LIN {X 0,Y 474.686,Z 291.355,A -85,B 0,C 180,E1 -7407.334,E2 -7407.334} C_VEL
LIN {X 0,Y 474.609,Z 291.36,A -85,B 0,C 180,E1 -7410.23,E2 -7410.23} C_VEL
LIN {X 0,Y 474.639,Z 291.365,A -85,B 0,C 180,E1 -7413.22,E2 -7413.22} C_VEL
LIN {X 0,Y 474.588,Z 291.363,A -85,B 0,C 180,E1 -7416.323,E2 -7416.323} C_VEL
LIN {X 0,Y 474.631,Z 291.363,A -85,B 0,C 180,E1 -7419.647,E2 -7419.647} C_VEL
LIN {X 0,Y 474.618,Z 291.361,A -85,B 0,C 180,E1 -7422.934,E2 -7422.934} C_VEL
LIN {X 0,Y 474.609,Z 291.365,A -85,B 0,C 180,E1 -7425.894,E2 -7425.894} C_VEL
LIN {X 0,Y 474.631,Z 291.358,A -85,B 0,C 180,E1 -7429.04,E2 -7429.04} C_VEL
LIN {X 0,Y 474.613,Z 291.367,A -85,B 0,C 180,E1 -7431.703,E2 -7431.703} C_VEL
LIN {X 0,Y 474.628,Z 291.358,A -85,B 0,C 180,E1 -7434.725,E2 -7434.725} C_VEL
LIN {X 0,Y 474.639,Z 291.362,A -85,B 0,C 180,E1 -7437.787,E2 -7437.787} C_VEL
LIN {X 0,Y 474.627,Z 291.358,A -85,B 0,C 180,E1 -7440.884,E2 -7440.884} C_VEL
LIN {X 0,Y 474.657,Z 291.356,A -85,B 0,C 180,E1 -7443.627,E2 -7443.627} C_VEL
LIN {X 0,Y 474.638,Z 291.36,A -85,B 0,C 180,E1 -7446.641,E2 -7446.641} C_VEL
LIN {X 0,Y 474.658,Z 291.358,A -85,B 0,C 180,E1 -7450.089,E2 -7450.089} C_VEL
LIN {X 0,Y 474.657,Z 291.354,A -85,B 0,C 180,E1 -7451.665,E2 -7451.665} C_VEL
LIN {X 0,Y 473.993,Z 291.444,A -85,B 0,C 180,E1 -7452.374,E2 -7452.374} C_VEL
LIN {X 0,Y 471.142,Z 291.796,A -85,B 0,C 180,E1 -7453.526,E2 -7453.526} C_VEL
LIN {X 0,Y 468.727,Z 292.1,A -85,B 0,C 180,E1 -7454.454,E2 -7454.454} C_VEL
LIN {X 0,Y 467.686,Z 292.224,A -85,B 0,C 180,E1 -7455.171,E2 -7455.171} C_VEL
LIN {X 0,Y 467.599,Z 292.234,A -85,B 0,C 180,E1 -7455.414,E2 -7455.414} C_VEL
LIN {X 0,Y 467.653,Z 292.235,A -85,B 0,C 180,E1 -7458.733,E2 -7458.733} C_VEL
LIN {X 0,Y 467.671,Z 292.229,A -85,B 0,C 180,E1 -7461.356,E2 -7461.356} C_VEL
LIN {X 0,Y 467.766,Z 292.344,A -85,B 0,C 180,E1 -7464.313,E2 -7464.313} C_VEL
LIN {X 0,Y 468.704,Z 298.944,A -85,B 0,C 180,E1 -7465.699,E2 -7465.699} C_VEL
LIN {X 0,Y 468.406,Z 311.043,A -85,B 0,C 180,E1 -7468.104,E2 -7468.104} C_VEL
LIN {X 0,Y 471.308,Z 326.851,A -85,B 0,C 180,E1 -7468.452,E2 -7468.452} C_VEL
LIN {X 0,Y 470.486,Z 418.039,A -85,B 0,C 180,E1 -7469.865,E2 -7469.865} C_VEL
LIN {X 0,Y 470.214,Z 431.176,A -85,B 0,C 180,E1 -7470.24,E2 -7470.24} C_VEL
LIN {X 0,Y 469.922,Z 444.292,A -85,B 0,C 180,E1 -7470.802,E2 -7470.802} C_VEL
LIN {X 0,Y 469.502,Z 456.173,A -85,B 0,C 180,E1 -7471.5,E2 -7471.5} C_VEL
LIN {X 0,Y 468.934,Z 467.583,A -85,B 0,C 180,E1 -7472.361,E2 -7472.361} C_VEL
LIN {X 0,Y 468.432,Z 477.859,A -85,B 0,C 180,E1 -7473.332,E2 -7473.332} C_VEL
LIN {X 0,Y 468.034,Z 486.265,A -85,B 0,C 180,E1 -7474.304,E2 -7474.304} C_VEL
LIN {X 0,Y 467.605,Z 495.387,A -85,B 0,C 180,E1 -7475.605,E2 -7475.605} C_VEL
LIN {X 0,Y 467.327,Z 503.183,A -85,B 0,C 180,E1 -7476.996,E2 -7476.996} C_VEL
LIN {X 0,Y 467.054,Z 508.653,A -85,B 0,C 180,E1 -7478.217,E2 -7478.217} C_VEL
LIN {X 0,Y 466.859,Z 513.329,A -85,B 0,C 180,E1 -7479.53,E2 -7479.53} C_VEL
LIN {X 0,Y 466.774,Z 516.89,A -85,B 0,C 180,E1 -7480.847,E2 -7480.847} C_VEL
LIN {X 0,Y 466.656,Z 519.437,A -85,B 0,C 180,E1 -7482.17,E2 -7482.17} C_VEL
LIN {X 0,Y 466.575,Z 520.608,A -85,B 0,C 180,E1 -7483.057,E2 -7483.057} C_VEL
LIN {X 0,Y 466.55,Z 521.33,A -85,B 0,C 180,E1 -7483.945,E2 -7483.945} C_VEL
LIN {X 0,Y 466.612,Z 521.631,A -85,B 0,C 180,E1 -7485.431,E2 -7485.431} C_VEL
LIN {X 0,Y 466.524,Z 521.04,A -85,B 0,C 180,E1 -7486.631,E2 -7486.631} C_VEL
LIN {X 0,Y 466.586,Z 520.075,A -85,B 0,C 180,E1 -7487.531,E2 -7487.531} C_VEL
LIN {X 0,Y 466.672,Z 518.689,A -85,B 0,C 180,E1 -7488.435,E2 -7488.435} C_VEL
LIN {X 0,Y 466.786,Z 515.7,A -85,B 0,C 180,E1 -7489.8,E2 -7489.8} C_VEL
LIN {X 0,Y 466.941,Z 511.554,A -85,B 0,C 180,E1 -7491.174,E2 -7491.174} C_VEL
LIN {X 0,Y 467.176,Z 506.077,A -85,B 0,C 180,E1 -7492.556,E2 -7492.556} C_VEL
LIN {X 0,Y 467.518,Z 499.072,A -85,B 0,C 180,E1 -7493.945,E2 -7493.945} C_VEL
LIN {X 0,Y 467.901,Z 491.826,A -85,B 0,C 180,E1 -7495.106,E2 -7495.106} C_VEL
LIN {X 0,Y 468.344,Z 482.951,A -85,B 0,C 180,E1 -7496.273,E2 -7496.273} C_VEL
LIN {X 0,Y 468.855,Z 473.048,A -85,B 0,C 180,E1 -7497.325,E2 -7497.325} C_VEL
LIN {X 0,Y 469.363,Z 461.573,A -85,B 0,C 180,E1 -7498.3,E2 -7498.3} C_VEL
LIN {X 0,Y 469.901,Z 449.823,A -85,B 0,C 180,E1 -7499.081,E2 -7499.081} C_VEL
LIN {X 0,Y 470.273,Z 438.126,A -85,B 0,C 180,E1 -7499.671,E2 -7499.671} C_VEL
LIN {X 0,Y 470.613,Z 424.916,A -85,B 0,C 180,E1 -7500.145,E2 -7500.145} C_VEL
LIN {X 0,Y 470.839,Z 411.912,A -85,B 0,C 180,E1 -7500.431,E2 -7500.431} C_VEL
LIN {X 0,Y 471.52,Z 325.739,A -85,B 0,C 180,E1 -7501.764,E2 -7501.764} C_VEL
LIN {X 0,Y 468.523,Z 310.731,A -85,B 0,C 180,E1 -7502.149,E2 -7502.149} C_VEL
LIN {X 0,Y 468.717,Z 298.947,A -85,B 0,C 180,E1 -7504.445,E2 -7504.445} C_VEL
LIN {X 0,Y 467.528,Z 292.25,A -85,B 0,C 180,E1 -7505.833,E2 -7505.833} C_VEL
LIN {X 0,Y 467.53,Z 292.248,A -85,B 0,C 180,E1 -7509.148,E2 -7509.148} C_VEL
LIN {X 0,Y 467.547,Z 292.247,A -85,B 0,C 180,E1 -7511.404,E2 -7511.404} C_VEL
LIN {X 0,Y 467.552,Z 292.246,A -85,B 0,C 180,E1 -7515.051,E2 -7515.051} C_VEL
LIN {X 0,Y 467.55,Z 292.242,A -85,B 0,C 180,E1 -7518.724,E2 -7518.724} C_VEL
LIN {X 0,Y 467.53,Z 292.248,A -85,B 0,C 180,E1 -7521.952,E2 -7521.952} C_VEL
LIN {X 0,Y 467.54,Z 292.236,A -85,B 0,C 180,E1 -7525.165,E2 -7525.165} C_VEL
LIN {X 0,Y 467.569,Z 292.238,A -85,B 0,C 180,E1 -7528.259,E2 -7528.259} C_VEL
LIN {X 0,Y 467.54,Z 292.244,A -85,B 0,C 180,E1 -7531.248,E2 -7531.248} C_VEL
LIN {X 0,Y 467.565,Z 292.241,A -85,B 0,C 180,E1 -7534.158,E2 -7534.158} C_VEL
LIN {X 0,Y 467.561,Z 292.239,A -85,B 0,C 180,E1 -7536.995,E2 -7536.995} C_VEL
LIN {X 0,Y 467.607,Z 292.234,A -85,B 0,C 180,E1 -7539.777,E2 -7539.777} C_VEL
LIN {X 0,Y 467.581,Z 292.236,A -85,B 0,C 180,E1 -7542.506,E2 -7542.506} C_VEL
LIN {X 0,Y 467.586,Z 292.236,A -85,B 0,C 180,E1 -7545.196,E2 -7545.196} C_VEL
LIN {X 0,Y 467.641,Z 292.231,A -85,B 0,C 180,E1 -7547.854,E2 -7547.854} C_VEL
LIN {X 0,Y 467.666,Z 292.226,A -85,B 0,C 180,E1 -7551.357,E2 -7551.357} C_VEL
LIN {X 0,Y 467.705,Z 292.219,A -85,B 0,C 180,E1 -7553.962,E2 -7553.962} C_VEL
LIN {X 0,Y 467.843,Z 292.2,A -85,B 0,C 180,E1 -7557.417,E2 -7557.417} C_VEL
LIN {X 0,Y 467.865,Z 292.201,A -85,B 0,C 180,E1 -7560,E2 -7560} C_VEL
LIN {X 0,Y 467.844,Z 292.205,A -85,B 0,C 180,E1 -7562.583,E2 -7562.583} C_VEL
LIN {X 0,Y 467.721,Z 292.22,A -85,B 0,C 180,E1 -7566.038,E2 -7566.038} C_VEL
LIN {X 0,Y 467.668,Z 292.226,A -85,B 0,C 180,E1 -7568.643,E2 -7568.643} C_VEL
LIN {X 0,Y 467.643,Z 292.229,A -85,B 0,C 180,E1 -7572.146,E2 -7572.146} C_VEL
LIN {X 0,Y 467.625,Z 292.231,A -85,B 0,C 180,E1 -7575.696,E2 -7575.696} C_VEL
LIN {X 0,Y 467.604,Z 292.235,A -85,B 0,C 180,E1 -7578.765,E2 -7578.765} C_VEL
LIN {X 0,Y 467.568,Z 292.243,A -85,B 0,C 180,E1 -7581.269,E2 -7581.269} C_VEL
LIN {X 0,Y 467.56,Z 292.236,A -85,B 0,C 180,E1 -7583.944,E2 -7583.944} C_VEL
LIN {X 0,Y 467.616,Z 292.237,A -85,B 0,C 180,E1 -7586.801,E2 -7586.801} C_VEL
LIN {X 0,Y 467.577,Z 292.24,A -85,B 0,C 180,E1 -7589.737,E2 -7589.737} C_VEL
LIN {X 0,Y 467.573,Z 292.237,A -85,B 0,C 180,E1 -7592.759,E2 -7592.759} C_VEL
LIN {X 0,Y 467.547,Z 292.243,A -85,B 0,C 180,E1 -7595.891,E2 -7595.891} C_VEL
LIN {X 0,Y 467.607,Z 292.239,A -85,B 0,C 180,E1 -7599.143,E2 -7599.143} C_VEL
LIN {X 0,Y 467.577,Z 292.237,A -85,B 0,C 180,E1 -7602.568,E2 -7602.568} C_VEL
LIN {X 0,Y 467.563,Z 292.24,A -85,B 0,C 180,E1 -7605.055,E2 -7605.055} C_VEL
LIN {X 0,Y 467.617,Z 292.235,A -85,B 0,C 180,E1 -7607.445,E2 -7607.445} C_VEL
LIN {X 0,Y 467.593,Z 292.234,A -85,B 0,C 180,E1 -7610.859,E2 -7610.859} C_VEL
LIN {X 0,Y 467.557,Z 292.245,A -85,B 0,C 180,E1 -7614.262,E2 -7614.262} C_VEL
LIN {X 0,Y 467.577,Z 292.24,A -85,B 0,C 180,E1 -7617.322,E2 -7617.322} C_VEL
LIN {X 0,Y 467.566,Z 292.242,A -85,B 0,C 180,E1 -7620.669,E2 -7620.669} C_VEL
LIN {X 0,Y 467.651,Z 292.234,A -85,B 0,C 180,E1 -7623.805,E2 -7623.805} C_VEL
LIN {X 0,Y 469.721,Z 302.869,A -85,B 0,C 180,E1 -7625.88,E2 -7625.88} C_VEL
LIN {X 0,Y 469.887,Z 307.145,A -85,B 0,C 180,E1 -7626.651,E2 -7626.651} C_VEL
LIN {X 0,Y 469.041,Z 325.461,A -85,B 0,C 180,E1 -7629.843,E2 -7629.843} C_VEL
LIN {X 0,Y 468.324,Z 343.295,A -85,B 0,C 180,E1 -7632.901,E2 -7632.901} C_VEL
LIN {X 0,Y 471.288,Z 362.293,A -85,B 0,C 180,E1 -7633.33,E2 -7633.33} C_VEL
LIN {X 0,Y 470.632,Z 452.171,A -85,B 0,C 180,E1 -7634.742,E2 -7634.742} C_VEL
LIN {X 0,Y 470.231,Z 465.287,A -85,B 0,C 180,E1 -7635.116,E2 -7635.116} C_VEL
LIN {X 0,Y 469.711,Z 477.936,A -85,B 0,C 180,E1 -7635.653,E2 -7635.653} C_VEL
LIN {X 0,Y 469.259,Z 489.997,A -85,B 0,C 180,E1 -7636.358,E2 -7636.358} C_VEL
LIN {X 0,Y 468.677,Z 501.749,A -85,B 0,C 180,E1 -7637.243,E2 -7637.243} C_VEL
LIN {X 0,Y 468.177,Z 512.937,A -85,B 0,C 180,E1 -7638.309,E2 -7638.309} C_VEL
LIN {X 0,Y 467.726,Z 522.081,A -85,B 0,C 180,E1 -7639.395,E2 -7639.395} C_VEL
LIN {X 0,Y 467.289,Z 531.006,A -85,B 0,C 180,E1 -7640.697,E2 -7640.697} C_VEL
LIN {X 0,Y 467.01,Z 538.19,A -85,B 0,C 180,E1 -7642,E2 -7642} C_VEL
LIN {X 0,Y 466.858,Z 543.046,A -85,B 0,C 180,E1 -7643.084,E2 -7643.084} C_VEL
LIN {X 0,Y 466.76,Z 547.769,A -85,B 0,C 180,E1 -7644.385,E2 -7644.385} C_VEL
LIN {X 0,Y 466.647,Z 551.376,A -85,B 0,C 180,E1 -7645.683,E2 -7645.683} C_VEL
LIN {X 0,Y 466.689,Z 553.239,A -85,B 0,C 180,E1 -7646.548,E2 -7646.548} C_VEL
LIN {X 0,Y 466.661,Z 554.634,A -85,B 0,C 180,E1 -7647.412,E2 -7647.412} C_VEL
LIN {X 0,Y 466.619,Z 556.239,A -85,B 0,C 180,E1 -7649.138,E2 -7649.138} C_VEL
LIN {X 0,Y 466.601,Z 556.45,A -85,B 0,C 180,E1 -7650.001,E2 -7650.001} C_VEL
LIN {X 0,Y 466.619,Z 556.229,A -85,B 0,C 180,E1 -7650.864,E2 -7650.864} C_VEL
LIN {X 0,Y 466.662,Z 554.617,A -85,B 0,C 180,E1 -7652.591,E2 -7652.591} C_VEL
LIN {X 0,Y 466.69,Z 553.208,A -85,B 0,C 180,E1 -7653.455,E2 -7653.455} C_VEL
LIN {X 0,Y 466.69,Z 550.25,A -85,B 0,C 180,E1 -7654.752,E2 -7654.752} C_VEL
LIN {X 0,Y 466.752,Z 546.245,A -85,B 0,C 180,E1 -7656.051,E2 -7656.051} C_VEL
LIN {X 0,Y 466.944,Z 540.078,A -85,B 0,C 180,E1 -7657.569,E2 -7657.569} C_VEL
LIN {X 0,Y 467.176,Z 533.344,A -85,B 0,C 180,E1 -7658.871,E2 -7658.871} C_VEL
LIN {X 0,Y 467.504,Z 524.988,A -85,B 0,C 180,E1 -7660.175,E2 -7660.175} C_VEL
LIN {X 0,Y 467.954,Z 516.396,A -85,B 0,C 180,E1 -7661.26,E2 -7661.26} C_VEL
LIN {X 0,Y 468.443,Z 506.232,A -85,B 0,C 180,E1 -7662.304,E2 -7662.304} C_VEL
LIN {X 0,Y 468.889,Z 495.273,A -85,B 0,C 180,E1 -7663.214,E2 -7663.214} C_VEL
LIN {X 0,Y 469.398,Z 483.688,A -85,B 0,C 180,E1 -7663.972,E2 -7663.972} C_VEL
LIN {X 0,Y 469.845,Z 471.654,A -85,B 0,C 180,E1 -7664.566,E2 -7664.566} C_VEL
LIN {X 0,Y 470.282,Z 458.632,A -85,B 0,C 180,E1 -7665.023,E2 -7665.023} C_VEL
LIN {X 0,Y 470.471,Z 446.371,A -85,B 0,C 180,E1 -7665.294,E2 -7665.294} C_VEL
LIN {X 0,Y 471.081,Z 362.542,A -85,B 0,C 180,E1 -7666.579,E2 -7666.579} C_VEL
LIN {X 0,Y 468.245,Z 343.636,A -85,B 0,C 180,E1 -7666.969,E2 -7666.969} C_VEL
LIN {X 0,Y 468.944,Z 326.257,A -85,B 0,C 180,E1 -7669.936,E2 -7669.936} C_VEL
LIN {X 0,Y 469.786,Z 306.459,A -85,B 0,C 180,E1 -7673.357,E2 -7673.357} C_VEL
LIN {X 0,Y 469.594,Z 302.376,A -85,B 0,C 180,E1 -7674.085,E2 -7674.085} C_VEL
LIN {X 0,Y 467.65,Z 292.236,A -85,B 0,C 180,E1 -7676.018,E2 -7676.018} C_VEL
LIN {X 0,Y 467.58,Z 292.239,A -85,B 0,C 180,E1 -7678.75,E2 -7678.75} C_VEL
LIN {X 0,Y 467.588,Z 292.237,A -85,B 0,C 180,E1 -7681.741,E2 -7681.741} C_VEL
LIN {X 0,Y 467.564,Z 292.24,A -85,B 0,C 180,E1 -7684.834,E2 -7684.834} C_VEL
LIN {X 0,Y 467.57,Z 292.241,A -85,B 0,C 180,E1 -7688.045,E2 -7688.045} C_VEL
LIN {X 0,Y 467.584,Z 292.236,A -85,B 0,C 180,E1 -7691.277,E2 -7691.277} C_VEL
LIN {X 0,Y 467.555,Z 292.239,A -85,B 0,C 180,E1 -7693.821,E2 -7693.821} C_VEL
LIN {X 0,Y 467.56,Z 292.241,A -85,B 0,C 180,E1 -7696.256,E2 -7696.256} C_VEL
LIN {X 0,Y 467.584,Z 292.244,A -85,B 0,C 180,E1 -7698.724,E2 -7698.724} C_VEL
LIN {X 0,Y 467.57,Z 292.237,A -85,B 0,C 180,E1 -7701.956,E2 -7701.956} C_VEL
LIN {X 0,Y 467.564,Z 292.244,A -85,B 0,C 180,E1 -7705.167,E2 -7705.167} C_VEL
LIN {X 0,Y 467.584,Z 292.235,A -85,B 0,C 180,E1 -7708.26,E2 -7708.26} C_VEL
LIN {X 0,Y 467.583,Z 292.243,A -85,B 0,C 180,E1 -7711.251,E2 -7711.251} C_VEL
LIN {X 0,Y 467.607,Z 292.232,A -85,B 0,C 180,E1 -7714.16,E2 -7714.16} C_VEL
LIN {X 0,Y 467.583,Z 292.239,A -85,B 0,C 180,E1 -7716.996,E2 -7716.996} C_VEL
LIN {X 0,Y 467.628,Z 292.234,A -85,B 0,C 180,E1 -7719.777,E2 -7719.777} C_VEL
LIN {X 0,Y 467.603,Z 292.233,A -85,B 0,C 180,E1 -7722.506,E2 -7722.506} C_VEL
LIN {X 0,Y 467.611,Z 292.235,A -85,B 0,C 180,E1 -7725.196,E2 -7725.196} C_VEL
LIN {X 0,Y 467.662,Z 292.232,A -85,B 0,C 180,E1 -7727.855,E2 -7727.855} C_VEL
LIN {X 0,Y 467.684,Z 292.225,A -85,B 0,C 180,E1 -7731.357,E2 -7731.357} C_VEL
LIN {X 0,Y 467.725,Z 292.226,A -85,B 0,C 180,E1 -7733.962,E2 -7733.962} C_VEL
LIN {X 0,Y 467.863,Z 292.202,A -85,B 0,C 180,E1 -7737.417,E2 -7737.417} C_VEL
LIN {X 0,Y 467.885,Z 292.205,A -85,B 0,C 180,E1 -7740,E2 -7740} C_VEL
LIN {X 0,Y 467.862,Z 292.204,A -85,B 0,C 180,E1 -7742.583,E2 -7742.583} C_VEL
LIN {X 0,Y 467.738,Z 292.221,A -85,B 0,C 180,E1 -7746.037,E2 -7746.037} C_VEL
LIN {X 0,Y 467.674,Z 292.229,A -85,B 0,C 180,E1 -7748.643,E2 -7748.643} C_VEL
LIN {X 0,Y 467.661,Z 292.229,A -85,B 0,C 180,E1 -7752.145,E2 -7752.145} C_VEL
LIN {X 0,Y 467.644,Z 292.228,A -85,B 0,C 180,E1 -7755.695,E2 -7755.695} C_VEL
LIN {X 0,Y 467.627,Z 292.232,A -85,B 0,C 180,E1 -7759.307,E2 -7759.307} C_VEL
LIN {X 0,Y 467.539,Z 292.241,A -85,B 0,C 180,E1 -7762.073,E2 -7762.073} C_VEL
LIN {X 0,Y 467.608,Z 292.241,A -85,B 0,C 180,E1 -7764.887,E2 -7764.887} C_VEL
LIN {X 0,Y 467.625,Z 292.231,A -85,B 0,C 180,E1 -7767.769,E2 -7767.769} C_VEL
LIN {X 0,Y 467.572,Z 292.245,A -85,B 0,C 180,E1 -7771.044,E2 -7771.044} C_VEL
LIN {X 0,Y 467.592,Z 292.234,A -85,B 0,C 180,E1 -7774.242,E2 -7774.242} C_VEL
LIN {X 0,Y 467.547,Z 292.247,A -85,B 0,C 180,E1 -7777.185,E2 -7777.185} C_VEL
LIN {X 0,Y 467.582,Z 292.236,A -85,B 0,C 180,E1 -7780.264,E2 -7780.264} C_VEL
LIN {X 0,Y 467.591,Z 292.234,A -85,B 0,C 180,E1 -7782.566,E2 -7782.566} C_VEL
LIN {X 0,Y 467.57,Z 292.239,A -85,B 0,C 180,E1 -7785.052,E2 -7785.052} C_VEL
LIN {X 0,Y 467.593,Z 292.24,A -85,B 0,C 180,E1 -7787.439,E2 -7787.439} C_VEL
LIN {X 0,Y 467.563,Z 292.238,A -85,B 0,C 180,E1 -7790.852,E2 -7790.852} C_VEL
LIN {X 0,Y 467.563,Z 292.241,A -85,B 0,C 180,E1 -7794.26,E2 -7794.26} C_VEL
LIN {X 0,Y 467.585,Z 292.236,A -85,B 0,C 180,E1 -7797.32,E2 -7797.32} C_VEL
LIN {X 0,Y 467.573,Z 292.238,A -85,B 0,C 180,E1 -7800.667,E2 -7800.667} C_VEL
LIN {X 0,Y 467.616,Z 292.231,A -85,B 0,C 180,E1 -7803.199,E2 -7803.199} C_VEL
LIN {X 0,Y 467.594,Z 292.24,A -85,B 0,C 180,E1 -7806.468,E2 -7806.468} C_VEL
LIN {X 0,Y 467.626,Z 292.231,A -85,B 0,C 180,E1 -7809.776,E2 -7809.776} C_VEL
LIN {X 0,Y 467.609,Z 292.241,A -85,B 0,C 180,E1 -7812.506,E2 -7812.506} C_VEL
LIN {X 0,Y 467.599,Z 292.234,A -85,B 0,C 180,E1 -7815.414,E2 -7815.414} C_VEL
LIN {X 0,Y 466.928,Z 292.321,A -85,B 0,C 180,E1 -7816.133,E2 -7816.133} C_VEL
LIN {X 0,Y 464.085,Z 292.673,A -85,B 0,C 180,E1 -7817.302,E2 -7817.302} C_VEL
LIN {X 0,Y 461.686,Z 292.973,A -85,B 0,C 180,E1 -7818.244,E2 -7818.244} C_VEL
LIN {X 0,Y 460.658,Z 293.103,A -85,B 0,C 180,E1 -7818.971,E2 -7818.971} C_VEL
LIN {X 0,Y 460.576,Z 293.109,A -85,B 0,C 180,E1 -7819.218,E2 -7819.218} C_VEL
LIN {X 0,Y 460.691,Z 293.102,A -85,B 0,C 180,E1 -7822.566,E2 -7822.566} C_VEL
LIN {X 0,Y 460.698,Z 293.153,A -85,B 0,C 180,E1 -7824.143,E2 -7824.143} C_VEL
LIN {X 0,Y 461.745,Z 300.164,A -85,B 0,C 180,E1 -7825.634,E2 -7825.634} C_VEL
LIN {X 0,Y 461.437,Z 311.165,A -85,B 0,C 180,E1 -7827.862,E2 -7827.862} C_VEL
LIN {X 0,Y 464.399,Z 326.503,A -85,B 0,C 180,E1 -7828.211,E2 -7828.211} C_VEL
LIN {X 0,Y 463.6,Z 418.943,A -85,B 0,C 180,E1 -7829.673,E2 -7829.673} C_VEL
LIN {X 0,Y 463.311,Z 431.88,A -85,B 0,C 180,E1 -7830.053,E2 -7830.053} C_VEL
LIN {X 0,Y 463.032,Z 444.33,A -85,B 0,C 180,E1 -7830.597,E2 -7830.597} C_VEL
LIN {X 0,Y 462.583,Z 456.292,A -85,B 0,C 180,E1 -7831.305,E2 -7831.305} C_VEL
LIN {X 0,Y 462.007,Z 467.734,A -85,B 0,C 180,E1 -7832.178,E2 -7832.178} C_VEL
LIN {X 0,Y 461.453,Z 478.048,A -85,B 0,C 180,E1 -7833.164,E2 -7833.164} C_VEL
LIN {X 0,Y 461.033,Z 486.476,A -85,B 0,C 180,E1 -7834.151,E2 -7834.151} C_VEL
LIN {X 0,Y 460.586,Z 495.616,A -85,B 0,C 180,E1 -7835.471,E2 -7835.471} C_VEL
LIN {X 0,Y 460.29,Z 502.846,A -85,B 0,C 180,E1 -7836.769,E2 -7836.769} C_VEL
LIN {X 0,Y 460.059,Z 507.991,A -85,B 0,C 180,E1 -7837.901,E2 -7837.901} C_VEL
LIN {X 0,Y 459.81,Z 512.864,A -85,B 0,C 180,E1 -7839.234,E2 -7839.234} C_VEL
LIN {X 0,Y 459.718,Z 516.605,A -85,B 0,C 180,E1 -7840.569,E2 -7840.569} C_VEL
LIN {X 0,Y 459.621,Z 519.256,A -85,B 0,C 180,E1 -7841.871,E2 -7841.871} C_VEL
LIN {X 0,Y 459.481,Z 521.074,A -85,B 0,C 180,E1 -7843.262,E2 -7843.262} C_VEL
LIN {X 0,Y 459.469,Z 521.716,A -85,B 0,C 180,E1 -7844.165,E2 -7844.165} C_VEL
LIN {X 0,Y 459.52,Z 521.884,A -85,B 0,C 180,E1 -7845.521,E2 -7845.521} C_VEL
LIN {X 0,Y 459.449,Z 521.102,A -85,B 0,C 180,E1 -7846.894,E2 -7846.894} C_VEL
LIN {X 0,Y 459.599,Z 518.882,A -85,B 0,C 180,E1 -7848.545,E2 -7848.545} C_VEL
LIN {X 0,Y 459.761,Z 515.355,A -85,B 0,C 180,E1 -7850.115,E2 -7850.115} C_VEL
LIN {X 0,Y 459.921,Z 510.995,A -85,B 0,C 180,E1 -7851.513,E2 -7851.513} C_VEL
LIN {X 0,Y 460.209,Z 505.305,A -85,B 0,C 180,E1 -7852.917,E2 -7852.917} C_VEL
LIN {X 0,Y 460.573,Z 498.069,A -85,B 0,C 180,E1 -7854.329,E2 -7854.329} C_VEL
LIN {X 0,Y 461.048,Z 489.45,A -85,B 0,C 180,E1 -7855.659,E2 -7855.659} C_VEL
LIN {X 0,Y 461.547,Z 480.205,A -85,B 0,C 180,E1 -7856.813,E2 -7856.813} C_VEL
LIN {X 0,Y 462.05,Z 470.897,A -85,B 0,C 180,E1 -7857.761,E2 -7857.761} C_VEL
LIN {X 0,Y 462.608,Z 459.799,A -85,B 0,C 180,E1 -7858.676,E2 -7858.676} C_VEL
LIN {X 0,Y 463.136,Z 448.139,A -85,B 0,C 180,E1 -7859.423,E2 -7859.423} C_VEL
LIN {X 0,Y 463.549,Z 435.864,A -85,B 0,C 180,E1 -7860.019,E2 -7860.019} C_VEL
LIN {X 0,Y 463.847,Z 423.53,A -85,B 0,C 180,E1 -7860.442,E2 -7860.442} C_VEL
LIN {X 0,Y 464.086,Z 408.879,A -85,B 0,C 180,E1 -7860.734,E2 -7860.734} C_VEL
LIN {X 0,Y 464.733,Z 326.376,A -85,B 0,C 180,E1 -7862.032,E2 -7862.032} C_VEL
LIN {X 0,Y 461.613,Z 310.999,A -85,B 0,C 180,E1 -7862.439,E2 -7862.439} C_VEL
LIN {X 0,Y 461.704,Z 299.479,A -85,B 0,C 180,E1 -7864.717,E2 -7864.717} C_VEL
LIN {X 0,Y 460.466,Z 293.13,A -85,B 0,C 180,E1 -7866.084,E2 -7866.084} C_VEL
LIN {X 0,Y 460.479,Z 293.126,A -85,B 0,C 180,E1 -7868.888,E2 -7868.888} C_VEL
LIN {X 0,Y 460.49,Z 293.127,A -85,B 0,C 180,E1 -7871.597,E2 -7871.597} C_VEL
LIN {X 0,Y 460.499,Z 293.121,A -85,B 0,C 180,E1 -7874.588,E2 -7874.588} C_VEL
LIN {X 0,Y 460.478,Z 293.127,A -85,B 0,C 180,E1 -7877.814,E2 -7877.814} C_VEL
LIN {X 0,Y 460.497,Z 293.122,A -85,B 0,C 180,E1 -7880.134,E2 -7880.134} C_VEL
LIN {X 0,Y 460.451,Z 293.126,A -85,B 0,C 180,E1 -7883.468,E2 -7883.468} C_VEL
LIN {X 0,Y 460.506,Z 293.119,A -85,B 0,C 180,E1 -7886.673,E2 -7886.673} C_VEL
LIN {X 0,Y 460.494,Z 293.126,A -85,B 0,C 180,E1 -7889.759,E2 -7889.759} C_VEL
LIN {X 0,Y 460.518,Z 293.117,A -85,B 0,C 180,E1 -7892.753,E2 -7892.753} C_VEL
LIN {X 0,Y 460.508,Z 293.12,A -85,B 0,C 180,E1 -7895.666,E2 -7895.666} C_VEL
LIN {X 0,Y 460.507,Z 293.115,A -85,B 0,C 180,E1 -7898.578,E2 -7898.578} C_VEL
LIN {X 0,Y 460.571,Z 293.111,A -85,B 0,C 180,E1 -7901.31,E2 -7901.31} C_VEL
LIN {X 0,Y 460.589,Z 293.11,A -85,B 0,C 180,E1 -7904.059,E2 -7904.059} C_VEL
LIN {X 0,Y 460.594,Z 293.107,A -85,B 0,C 180,E1 -7907.666,E2 -7907.666} C_VEL
LIN {X 0,Y 460.613,Z 293.104,A -85,B 0,C 180,E1 -7911.224,E2 -7911.224} C_VEL
LIN {X 0,Y 460.669,Z 293.094,A -85,B 0,C 180,E1 -7913.87,E2 -7913.87} C_VEL
LIN {X 0,Y 460.785,Z 293.079,A -85,B 0,C 180,E1 -7917.378,E2 -7917.378} C_VEL
LIN {X 0,Y 460.836,Z 293.077,A -85,B 0,C 180,E1 -7920,E2 -7920} C_VEL
LIN {X 0,Y 460.785,Z 293.083,A -85,B 0,C 180,E1 -7922.623,E2 -7922.623} C_VEL
LIN {X 0,Y 460.687,Z 293.097,A -85,B 0,C 180,E1 -7926.13,E2 -7926.13} C_VEL
LIN {X 0,Y 460.615,Z 293.105,A -85,B 0,C 180,E1 -7928.777,E2 -7928.777} C_VEL
LIN {X 0,Y 460.599,Z 293.109,A -85,B 0,C 180,E1 -7932.445,E2 -7932.445} C_VEL
LIN {X 0,Y 460.586,Z 293.108,A -85,B 0,C 180,E1 -7935.998,E2 -7935.998} C_VEL
LIN {X 0,Y 460.557,Z 293.113,A -85,B 0,C 180,E1 -7938.902,E2 -7938.902} C_VEL
LIN {X 0,Y 460.503,Z 293.12,A -85,B 0,C 180,E1 -7941.486,E2 -7941.486} C_VEL
LIN {X 0,Y 460.53,Z 293.112,A -85,B 0,C 180,E1 -7944.333,E2 -7944.333} C_VEL
LIN {X 0,Y 460.572,Z 293.112,A -85,B 0,C 180,E1 -7947.244,E2 -7947.244} C_VEL
LIN {X 0,Y 460.519,Z 293.117,A -85,B 0,C 180,E1 -7950.24,E2 -7950.24} C_VEL
LIN {X 0,Y 460.519,Z 293.123,A -85,B 0,C 180,E1 -7953.326,E2 -7953.326} C_VEL
LIN {X 0,Y 460.47,Z 293.122,A -85,B 0,C 180,E1 -7956.53,E2 -7956.53} C_VEL
LIN {X 0,Y 460.567,Z 293.115,A -85,B 0,C 180,E1 -7959.859,E2 -7959.859} C_VEL
LIN {X 0,Y 460.508,Z 293.118,A -85,B 0,C 180,E1 -7962.902,E2 -7962.902} C_VEL
LIN {X 0,Y 460.516,Z 293.115,A -85,B 0,C 180,E1 -7965.83,E2 -7965.83} C_VEL
LIN {X 0,Y 460.536,Z 293.116,A -85,B 0,C 180,E1 -7968.992,E2 -7968.992} C_VEL
LIN {X 0,Y 460.533,Z 293.116,A -85,B 0,C 180,E1 -7971.27,E2 -7971.27} C_VEL
LIN {X 0,Y 460.507,Z 293.121,A -85,B 0,C 180,E1 -7974.556,E2 -7974.556} C_VEL
LIN {X 0,Y 460.526,Z 293.123,A -85,B 0,C 180,E1 -7977.717,E2 -7977.717} C_VEL
LIN {X 0,Y 460.536,Z 293.118,A -85,B 0,C 180,E1 -7980.771,E2 -7980.771} C_VEL
LIN {X 0,Y 460.622,Z 293.272,A -85,B 0,C 180,E1 -7983.618,E2 -7983.618} C_VEL
LIN {X 0,Y 462.827,Z 304.413,A -85,B 0,C 180,E1 -7985.797,E2 -7985.797} C_VEL
LIN {X 0,Y 462.972,Z 308.34,A -85,B 0,C 180,E1 -7986.519,E2 -7986.519} C_VEL
LIN {X 0,Y 462.08,Z 326.655,A -85,B 0,C 180,E1 -7989.758,E2 -7989.758} C_VEL
LIN {X 0,Y 461.369,Z 343.062,A -85,B 0,C 180,E1 -7992.62,E2 -7992.62} C_VEL
LIN {X 0,Y 464.544,Z 363.97,A -85,B 0,C 180,E1 -7993.089,E2 -7993.089} C_VEL
LIN {X 0,Y 463.843,Z 451.619,A -85,B 0,C 180,E1 -7994.485,E2 -7994.485} C_VEL
LIN {X 0,Y 463.429,Z 464.827,A -85,B 0,C 180,E1 -7994.865,E2 -7994.865} C_VEL
LIN {X 0,Y 462.86,Z 478.082,A -85,B 0,C 180,E1 -7995.436,E2 -7995.436} C_VEL
LIN {X 0,Y 462.367,Z 490.017,A -85,B 0,C 180,E1 -7996.15,E2 -7996.15} C_VEL
LIN {X 0,Y 461.792,Z 500.723,A -85,B 0,C 180,E1 -7996.965,E2 -7996.965} C_VEL
LIN {X 0,Y 461.28,Z 511.808,A -85,B 0,C 180,E1 -7998.02,E2 -7998.02} C_VEL
LIN {X 0,Y 460.794,Z 520.272,A -85,B 0,C 180,E1 -7999.011,E2 -7999.011} C_VEL
LIN {X 0,Y 460.309,Z 529.459,A -85,B 0,C 180,E1 -8000.333,E2 -8000.333} C_VEL
LIN {X 0,Y 460,Z 536.87,A -85,B 0,C 180,E1 -8001.656,E2 -8001.656} C_VEL
LIN {X 0,Y 459.775,Z 542.83,A -85,B 0,C 180,E1 -8002.977,E2 -8002.977} C_VEL
LIN {X 0,Y 459.656,Z 547.542,A -85,B 0,C 180,E1 -8004.298,E2 -8004.298} C_VEL
LIN {X 0,Y 459.564,Z 551.141,A -85,B 0,C 180,E1 -8005.616,E2 -8005.616} C_VEL
LIN {X 0,Y 459.585,Z 552.995,A -85,B 0,C 180,E1 -8006.494,E2 -8006.494} C_VEL
LIN {X 0,Y 459.584,Z 554.385,A -85,B 0,C 180,E1 -8007.372,E2 -8007.372} C_VEL
LIN {X 0,Y 459.523,Z 555.981,A -85,B 0,C 180,E1 -8009.125,E2 -8009.125} C_VEL
LIN {X 0,Y 459.532,Z 556.186,A -85,B 0,C 180,E1 -8010.001,E2 -8010.001} C_VEL
LIN {X 0,Y 459.552,Z 555.958,A -85,B 0,C 180,E1 -8010.878,E2 -8010.878} C_VEL
LIN {X 0,Y 459.584,Z 554.336,A -85,B 0,C 180,E1 -8012.631,E2 -8012.631} C_VEL
LIN {X 0,Y 459.586,Z 552.917,A -85,B 0,C 180,E1 -8013.508,E2 -8013.508} C_VEL
LIN {X 0,Y 459.617,Z 549.951,A -85,B 0,C 180,E1 -8014.826,E2 -8014.826} C_VEL
LIN {X 0,Y 459.716,Z 544.886,A -85,B 0,C 180,E1 -8016.432,E2 -8016.432} C_VEL
LIN {X 0,Y 459.894,Z 538.732,A -85,B 0,C 180,E1 -8017.907,E2 -8017.907} C_VEL
LIN {X 0,Y 460.189,Z 531.755,A -85,B 0,C 180,E1 -8019.229,E2 -8019.229} C_VEL
LIN {X 0,Y 460.564,Z 523.002,A -85,B 0,C 180,E1 -8020.552,E2 -8020.552} C_VEL
LIN {X 0,Y 461.058,Z 514.04,A -85,B 0,C 180,E1 -8021.654,E2 -8021.654} C_VEL
LIN {X 0,Y 461.546,Z 504.309,A -85,B 0,C 180,E1 -8022.633,E2 -8022.633} C_VEL
LIN {X 0,Y 462.016,Z 493.31,A -85,B 0,C 180,E1 -8023.527,E2 -8023.527} C_VEL
LIN {X 0,Y 462.576,Z 481.107,A -85,B 0,C 180,E1 -8024.295,E2 -8024.295} C_VEL
LIN {X 0,Y 463.048,Z 468.338,A -85,B 0,C 180,E1 -8024.898,E2 -8024.898} C_VEL
LIN {X 0,Y 463.478,Z 455.671,A -85,B 0,C 180,E1 -8025.305,E2 -8025.305} C_VEL
LIN {X 0,Y 463.709,Z 439.528,A -85,B 0,C 180,E1 -8025.607,E2 -8025.607} C_VEL
LIN {X 0,Y 464.125,Z 362.39,A -85,B 0,C 180,E1 -8026.811,E2 -8026.811} C_VEL
LIN {X 0,Y 461.259,Z 343.25,A -85,B 0,C 180,E1 -8027.234,E2 -8027.234} C_VEL
LIN {X 0,Y 461.936,Z 327.178,A -85,B 0,C 180,E1 -8030.019,E2 -8030.019} C_VEL
LIN {X 0,Y 462.828,Z 307.357,A -85,B 0,C 180,E1 -8033.492,E2 -8033.492} C_VEL
LIN {X 0,Y 462.539,Z 303.123,A -85,B 0,C 180,E1 -8034.263,E2 -8034.263} C_VEL
LIN {X 0,Y 460.594,Z 293.114,A -85,B 0,C 180,E1 -8036.202,E2 -8036.202} C_VEL
LIN {X 0,Y 460.544,Z 293.115,A -85,B 0,C 180,E1 -8039.232,E2 -8039.232} C_VEL
LIN {X 0,Y 460.536,Z 293.121,A -85,B 0,C 180,E1 -8042.285,E2 -8042.285} C_VEL
LIN {X 0,Y 460.514,Z 293.116,A -85,B 0,C 180,E1 -8045.446,E2 -8045.446} C_VEL
LIN {X 0,Y 460.538,Z 293.115,A -85,B 0,C 180,E1 -8048.896,E2 -8048.896} C_VEL
LIN {X 0,Y 460.529,Z 293.118,A -85,B 0,C 180,E1 -8052.182,E2 -8052.182} C_VEL
LIN {X 0,Y 460.52,Z 293.116,A -85,B 0,C 180,E1 -8055.411,E2 -8055.411} C_VEL
LIN {X 0,Y 460.538,Z 293.117,A -85,B 0,C 180,E1 -8058.398,E2 -8058.398} C_VEL
LIN {X 0,Y 460.529,Z 293.117,A -85,B 0,C 180,E1 -8061.267,E2 -8061.267} C_VEL
LIN {X 0,Y 460.514,Z 293.119,A -85,B 0,C 180,E1 -8064.554,E2 -8064.554} C_VEL
LIN {X 0,Y 460.531,Z 293.115,A -85,B 0,C 180,E1 -8067.715,E2 -8067.715} C_VEL
LIN {X 0,Y 460.546,Z 293.116,A -85,B 0,C 180,E1 -8070.769,E2 -8070.769} C_VEL
LIN {X 0,Y 460.565,Z 293.112,A -85,B 0,C 180,E1 -8073.735,E2 -8073.735} C_VEL
LIN {X 0,Y 460.552,Z 293.112,A -85,B 0,C 180,E1 -8076.624,E2 -8076.624} C_VEL
LIN {X 0,Y 460.557,Z 293.119,A -85,B 0,C 180,E1 -8079.453,E2 -8079.453} C_VEL
LIN {X 0,Y 460.554,Z 293.112,A -85,B 0,C 180,E1 -8082.23,E2 -8082.23} C_VEL
LIN {X 0,Y 460.57,Z 293.11,A -85,B 0,C 180,E1 -8084.965,E2 -8084.965} C_VEL
LIN {X 0,Y 460.615,Z 293.104,A -85,B 0,C 180,E1 -8088.559,E2 -8088.559} C_VEL
LIN {X 0,Y 460.672,Z 293.101,A -85,B 0,C 180,E1 -8092.108,E2 -8092.108} C_VEL
LIN {X 0,Y 460.693,Z 293.094,A -85,B 0,C 180,E1 -8094.748,E2 -8094.748} C_VEL
LIN {X 0,Y 460.804,Z 293.081,A -85,B 0,C 180,E1 -8097.377,E2 -8097.377} C_VEL
LIN {X 0,Y 460.856,Z 293.081,A -85,B 0,C 180,E1 -8100,E2 -8100} C_VEL
LIN {X 0,Y 460.803,Z 293.083,A -85,B 0,C 180,E1 -8102.622,E2 -8102.622} C_VEL
LIN {X 0,Y 460.703,Z 293.099,A -85,B 0,C 180,E1 -8106.13,E2 -8106.13} C_VEL
LIN {X 0,Y 460.624,Z 293.106,A -85,B 0,C 180,E1 -8108.776,E2 -8108.776} C_VEL
LIN {X 0,Y 460.619,Z 293.111,A -85,B 0,C 180,E1 -8112.445,E2 -8112.445} C_VEL
LIN {X 0,Y 460.606,Z 293.106,A -85,B 0,C 180,E1 -8115.997,E2 -8115.997} C_VEL
LIN {X 0,Y 460.573,Z 293.109,A -85,B 0,C 180,E1 -8119.615,E2 -8119.615} C_VEL
LIN {X 0,Y 460.515,Z 293.119,A -85,B 0,C 180,E1 -8122.428,E2 -8122.428} C_VEL
LIN {X 0,Y 460.573,Z 293.109,A -85,B 0,C 180,E1 -8125.801,E2 -8125.801} C_VEL
LIN {X 0,Y 460.557,Z 293.111,A -85,B 0,C 180,E1 -8128.232,E2 -8128.232} C_VEL
LIN {X 0,Y 460.525,Z 293.121,A -85,B 0,C 180,E1 -8131.282,E2 -8131.282} C_VEL
LIN {X 0,Y 460.535,Z 293.114,A -85,B 0,C 180,E1 -8134.505,E2 -8134.505} C_VEL
LIN {X 0,Y 460.503,Z 293.122,A -85,B 0,C 180,E1 -8137.623,E2 -8137.623} C_VEL
LIN {X 0,Y 460.546,Z 293.112,A -85,B 0,C 180,E1 -8140.269,E2 -8140.269} C_VEL
LIN {X 0,Y 460.503,Z 293.124,A -85,B 0,C 180,E1 -8143.375,E2 -8143.375} C_VEL
LIN {X 0,Y 460.5,Z 293.118,A -85,B 0,C 180,E1 -8146.624,E2 -8146.624} C_VEL
LIN {X 0,Y 460.543,Z 293.122,A -85,B 0,C 180,E1 -8149.73,E2 -8149.73} C_VEL
LIN {X 0,Y 460.503,Z 293.118,A -85,B 0,C 180,E1 -8152.523,E2 -8152.523} C_VEL
LIN {X 0,Y 460.55,Z 293.116,A -85,B 0,C 180,E1 -8155.623,E2 -8155.623} C_VEL
LIN {X 0,Y 460.541,Z 293.113,A -85,B 0,C 180,E1 -8158.744,E2 -8158.744} C_VEL
LIN {X 0,Y 460.585,Z 293.115,A -85,B 0,C 180,E1 -8162.253,E2 -8162.253} C_VEL
LIN {X 0,Y 460.543,Z 293.115,A -85,B 0,C 180,E1 -8164.703,E2 -8164.703} C_VEL
LIN {X 0,Y 460.514,Z 293.116,A -85,B 0,C 180,E1 -8167.57,E2 -8167.57} C_VEL
LIN {X 0,Y 460.572,Z 293.117,A -85,B 0,C 180,E1 -8170.384,E2 -8170.384} C_VEL
LIN {X 0,Y 460.566,Z 293.111,A -85,B 0,C 180,E1 -8173.145,E2 -8173.145} C_VEL
LIN {X 0,Y 460.556,Z 293.111,A -85,B 0,C 180,E1 -8175.867,E2 -8175.867} C_VEL
LIN {X 0,Y 460.612,Z 293.111,A -85,B 0,C 180,E1 -8178.558,E2 -8178.558} C_VEL
LIN {X 0,Y 460.576,Z 293.109,A -85,B 0,C 180,E1 -8179.218,E2 -8179.218} C_VEL
LIN {X 0,Y 459.916,Z 293.191,A -85,B 0,C 180,E1 -8179.948,E2 -8179.948} C_VEL
LIN {X 0,Y 457.089,Z 293.549,A -85,B 0,C 180,E1 -8181.133,E2 -8181.133} C_VEL
LIN {X 0,Y 454.706,Z 293.85,A -85,B 0,C 180,E1 -8182.09,E2 -8182.09} C_VEL
LIN {X 0,Y 453.695,Z 293.975,A -85,B 0,C 180,E1 -8182.829,E2 -8182.829} C_VEL
LIN {X 0,Y 453.619,Z 293.983,A -85,B 0,C 180,E1 -8183.079,E2 -8183.079} C_VEL
LIN {X 0,Y 453.663,Z 294.077,A -85,B 0,C 180,E1 -8183.996,E2 -8183.996} C_VEL
LIN {X 0,Y 454.767,Z 301.367,A -85,B 0,C 180,E1 -8185.567,E2 -8185.567} C_VEL
LIN {X 0,Y 454.5,Z 311.383,A -85,B 0,C 180,E1 -8187.614,E2 -8187.614} C_VEL
LIN {X 0,Y 457.625,Z 327.961,A -85,B 0,C 180,E1 -8187.996,E2 -8187.996} C_VEL
LIN {X 0,Y 456.735,Z 418.419,A -85,B 0,C 180,E1 -8189.439,E2 -8189.439} C_VEL
LIN {X 0,Y 456.425,Z 431.394,A -85,B 0,C 180,E1 -8189.817,E2 -8189.817} C_VEL
LIN {X 0,Y 456.126,Z 444.366,A -85,B 0,C 180,E1 -8190.385,E2 -8190.385} C_VEL
LIN {X 0,Y 455.675,Z 456.387,A -85,B 0,C 180,E1 -8191.103,E2 -8191.103} C_VEL
LIN {X 0,Y 455.064,Z 467.864,A -85,B 0,C 180,E1 -8191.99,E2 -8191.99} C_VEL
LIN {X 0,Y 454.49,Z 478.199,A -85,B 0,C 180,E1 -8192.99,E2 -8192.99} C_VEL
LIN {X 0,Y 454.053,Z 486.645,A -85,B 0,C 180,E1 -8193.993,E2 -8193.993} C_VEL
LIN {X 0,Y 453.648,Z 494.445,A -85,B 0,C 180,E1 -8195.109,E2 -8195.109} C_VEL
LIN {X 0,Y 453.289,Z 502.321,A -85,B 0,C 180,E1 -8196.504,E2 -8196.504} C_VEL
LIN {X 0,Y 452.946,Z 509.119,A -85,B 0,C 180,E1 -8198.026,E2 -8198.026} C_VEL
LIN {X 0,Y 452.721,Z 513.812,A -85,B 0,C 180,E1 -8199.38,E2 -8199.38} C_VEL
LIN {X 0,Y 452.635,Z 517.384,A -85,B 0,C 180,E1 -8200.737,E2 -8200.737} C_VEL
LIN {X 0,Y 452.531,Z 519.657,A -85,B 0,C 180,E1 -8201.926,E2 -8201.926} C_VEL
LIN {X 0,Y 452.386,Z 521.536,A -85,B 0,C 180,E1 -8203.474,E2 -8203.474} C_VEL
LIN {X 0,Y 452.376,Z 522.092,A -85,B 0,C 180,E1 -8204.391,E2 -8204.391} C_VEL
LIN {X 0,Y 452.418,Z 522.139,A -85,B 0,C 180,E1 -8205.608,E2 -8205.608} C_VEL
LIN {X 0,Y 452.373,Z 521.17,A -85,B 0,C 180,E1 -8207.167,E2 -8207.167} C_VEL
LIN {X 0,Y 452.526,Z 519.058,A -85,B 0,C 180,E1 -8208.672,E2 -8208.672} C_VEL
LIN {X 0,Y 452.657,Z 516.264,A -85,B 0,C 180,E1 -8209.971,E2 -8209.971} C_VEL
LIN {X 0,Y 452.816,Z 512.192,A -85,B 0,C 180,E1 -8211.371,E2 -8211.371} C_VEL
LIN {X 0,Y 453.104,Z 506.677,A -85,B 0,C 180,E1 -8212.814,E2 -8212.814} C_VEL
LIN {X 0,Y 453.514,Z 499.7,A -85,B 0,C 180,E1 -8214.244,E2 -8214.244} C_VEL
LIN {X 0,Y 453.926,Z 492.474,A -85,B 0,C 180,E1 -8215.443,E2 -8215.443} C_VEL
LIN {X 0,Y 454.482,Z 483.647,A -85,B 0,C 180,E1 -8216.642,E2 -8216.642} C_VEL
LIN {X 0,Y 455.019,Z 473.904,A -85,B 0,C 180,E1 -8217.716,E2 -8217.716} C_VEL
LIN {X 0,Y 455.598,Z 462.85,A -85,B 0,C 180,E1 -8218.692,E2 -8218.692} C_VEL
LIN {X 0,Y 456.215,Z 450.728,A -85,B 0,C 180,E1 -8219.533,E2 -8219.533} C_VEL
LIN {X 0,Y 456.65,Z 439.236,A -85,B 0,C 180,E1 -8220.138,E2 -8220.138} C_VEL
LIN {X 0,Y 457.018,Z 426.417,A -85,B 0,C 180,E1 -8220.621,E2 -8220.621} C_VEL
LIN {X 0,Y 457.269,Z 413.73,A -85,B 0,C 180,E1 -8220.923,E2 -8220.923} C_VEL
LIN {X 0,Y 457.975,Z 327.037,A -85,B 0,C 180,E1 -8222.313,E2 -8222.313} C_VEL
LIN {X 0,Y 454.708,Z 311.384,A -85,B 0,C 180,E1 -8222.717,E2 -8222.717} C_VEL
LIN {X 0,Y 454.884,Z 301.951,A -85,B 0,C 180,E1 -8224.594,E2 -8224.594} C_VEL
LIN {X 0,Y 453.427,Z 294.007,A -85,B 0,C 180,E1 -8226.295,E2 -8226.295} C_VEL
LIN {X 0,Y 453.429,Z 294.006,A -85,B 0,C 180,E1 -8229.454,E2 -8229.454} C_VEL
LIN {X 0,Y 453.424,Z 294.005,A -85,B 0,C 180,E1 -8231.928,E2 -8231.928} C_VEL
LIN {X 0,Y 453.469,Z 293.998,A -85,B 0,C 180,E1 -8235.471,E2 -8235.471} C_VEL
LIN {X 0,Y 453.439,Z 294.001,A -85,B 0,C 180,E1 -8238.205,E2 -8238.205} C_VEL
LIN {X 0,Y 453.426,Z 294.002,A -85,B 0,C 180,E1 -8240.801,E2 -8240.801} C_VEL
LIN {X 0,Y 453.433,Z 293.994,A -85,B 0,C 180,E1 -8243.915,E2 -8243.915} C_VEL
LIN {X 0,Y 453.465,Z 293.998,A -85,B 0,C 180,E1 -8247.15,E2 -8247.15} C_VEL
LIN {X 0,Y 453.453,Z 293.999,A -85,B 0,C 180,E1 -8250.267,E2 -8250.267} C_VEL
LIN {X 0,Y 453.454,Z 293.998,A -85,B 0,C 180,E1 -8253.291,E2 -8253.291} C_VEL
LIN {X 0,Y 453.48,Z 293.998,A -85,B 0,C 180,E1 -8256.238,E2 -8256.238} C_VEL
LIN {X 0,Y 453.467,Z 293.991,A -85,B 0,C 180,E1 -8259.117,E2 -8259.117} C_VEL
LIN {X 0,Y 453.488,Z 293.999,A -85,B 0,C 180,E1 -8261.944,E2 -8261.944} C_VEL
LIN {X 0,Y 453.522,Z 293.989,A -85,B 0,C 180,E1 -8264.726,E2 -8264.726} C_VEL
LIN {X 0,Y 453.544,Z 293.987,A -85,B 0,C 180,E1 -8268.379,E2 -8268.379} C_VEL
LIN {X 0,Y 453.577,Z 293.981,A -85,B 0,C 180,E1 -8271.087,E2 -8271.087} C_VEL
LIN {X 0,Y 453.635,Z 293.97,A -85,B 0,C 180,E1 -8273.774,E2 -8273.774} C_VEL
LIN {X 0,Y 453.729,Z 293.958,A -85,B 0,C 180,E1 -8277.337,E2 -8277.337} C_VEL
LIN {X 0,Y 453.807,Z 293.952,A -85,B 0,C 180,E1 -8280,E2 -8280} C_VEL
LIN {X 0,Y 453.73,Z 293.961,A -85,B 0,C 180,E1 -8282.664,E2 -8282.664} C_VEL
LIN {X 0,Y 453.655,Z 293.974,A -85,B 0,C 180,E1 -8286.226,E2 -8286.226} C_VEL
LIN {X 0,Y 453.579,Z 293.981,A -85,B 0,C 180,E1 -8288.914,E2 -8288.914} C_VEL
LIN {X 0,Y 453.549,Z 293.989,A -85,B 0,C 180,E1 -8292.529,E2 -8292.529} C_VEL
LIN {X 0,Y 453.531,Z 293.988,A -85,B 0,C 180,E1 -8296.197,E2 -8296.197} C_VEL
LIN {X 0,Y 453.507,Z 293.991,A -85,B 0,C 180,E1 -8299.041,E2 -8299.041} C_VEL
LIN {X 0,Y 453.464,Z 293.995,A -85,B 0,C 180,E1 -8301.837,E2 -8301.837} C_VEL
LIN {X 0,Y 453.502,Z 293.99,A -85,B 0,C 180,E1 -8304.735,E2 -8304.735} C_VEL
LIN {X 0,Y 453.527,Z 293.983,A -85,B 0,C 180,E1 -8307.962,E2 -8307.962} C_VEL
LIN {X 0,Y 453.473,Z 293.997,A -85,B 0,C 180,E1 -8310.76,E2 -8310.76} C_VEL
LIN {X 0,Y 453.467,Z 293.998,A -85,B 0,C 180,E1 -8313.914,E2 -8313.914} C_VEL
LIN {X 0,Y 453.462,Z 294.001,A -85,B 0,C 180,E1 -8317.189,E2 -8317.189} C_VEL
LIN {X 0,Y 453.522,Z 293.994,A -85,B 0,C 180,E1 -8319.447,E2 -8319.447} C_VEL
LIN {X 0,Y 453.459,Z 293.997,A -85,B 0,C 180,E1 -8322.996,E2 -8322.996} C_VEL
LIN {X 0,Y 453.469,Z 293.992,A -85,B 0,C 180,E1 -8325.782,E2 -8325.782} C_VEL
LIN {X 0,Y 453.489,Z 293.995,A -85,B 0,C 180,E1 -8328.213,E2 -8328.213} C_VEL
LIN {X 0,Y 453.52,Z 293.987,A -85,B 0,C 180,E1 -8330.79,E2 -8330.79} C_VEL
LIN {X 0,Y 453.451,Z 294,A -85,B 0,C 180,E1 -8333.919,E2 -8333.919} C_VEL
LIN {X 0,Y 453.478,Z 293.995,A -85,B 0,C 180,E1 -8337.153,E2 -8337.153} C_VEL
LIN {X 0,Y 453.471,Z 293.999,A -85,B 0,C 180,E1 -8340.27,E2 -8340.27} C_VEL
LIN {X 0,Y 453.587,Z 294.107,A -85,B 0,C 180,E1 -8343.347,E2 -8343.347} C_VEL
LIN {X 0,Y 455.857,Z 305.669,A -85,B 0,C 180,E1 -8345.65,E2 -8345.65} C_VEL
LIN {X 0,Y 456.085,Z 309.571,A -85,B 0,C 180,E1 -8346.383,E2 -8346.383} C_VEL
LIN {X 0,Y 455.159,Z 326.543,A -85,B 0,C 180,E1 -8349.436,E2 -8349.436} C_VEL
LIN {X 0,Y 454.434,Z 342.777,A -85,B 0,C 180,E1 -8352.315,E2 -8352.315} C_VEL
LIN {X 0,Y 457.745,Z 363.806,A -85,B 0,C 180,E1 -8352.806,E2 -8352.806} C_VEL
LIN {X 0,Y 457.037,Z 451.085,A -85,B 0,C 180,E1 -8354.219,E2 -8354.219} C_VEL
LIN {X 0,Y 456.597,Z 464.367,A -85,B 0,C 180,E1 -8354.604,E2 -8354.604} C_VEL
LIN {X 0,Y 456.08,Z 477.111,A -85,B 0,C 180,E1 -8355.158,E2 -8355.158} C_VEL
LIN {X 0,Y 455.544,Z 488.453,A -85,B 0,C 180,E1 -8355.825,E2 -8355.825} C_VEL
LIN {X 0,Y 454.861,Z 500.637,A -85,B 0,C 180,E1 -8356.757,E2 -8356.757} C_VEL
LIN {X 0,Y 454.325,Z 511.735,A -85,B 0,C 180,E1 -8357.834,E2 -8357.834} C_VEL
LIN {X 0,Y 453.699,Z 521.807,A -85,B 0,C 180,E1 -8359.063,E2 -8359.063} C_VEL
LIN {X 0,Y 453.199,Z 530.677,A -85,B 0,C 180,E1 -8360.405,E2 -8360.405} C_VEL
LIN {X 0,Y 452.903,Z 537.807,A -85,B 0,C 180,E1 -8361.749,E2 -8361.749} C_VEL
LIN {X 0,Y 452.634,Z 544.318,A -85,B 0,C 180,E1 -8363.315,E2 -8363.315} C_VEL
LIN {X 0,Y 452.563,Z 548.627,A -85,B 0,C 180,E1 -8364.655,E2 -8364.655} C_VEL
LIN {X 0,Y 452.486,Z 550.913,A -85,B 0,C 180,E1 -8365.547,E2 -8365.547} C_VEL
LIN {X 0,Y 452.481,Z 552.754,A -85,B 0,C 180,E1 -8366.439,E2 -8366.439} C_VEL
LIN {X 0,Y 452.507,Z 554.139,A -85,B 0,C 180,E1 -8367.331,E2 -8367.331} C_VEL
LIN {X 0,Y 452.43,Z 555.724,A -85,B 0,C 180,E1 -8369.111,E2 -8369.111} C_VEL
LIN {X 0,Y 452.465,Z 555.921,A -85,B 0,C 180,E1 -8370.001,E2 -8370.001} C_VEL
LIN {X 0,Y 452.457,Z 555.065,A -85,B 0,C 180,E1 -8371.782,E2 -8371.782} C_VEL
LIN {X 0,Y 452.508,Z 554.054,A -85,B 0,C 180,E1 -8372.672,E2 -8372.672} C_VEL
LIN {X 0,Y 452.484,Z 552.624,A -85,B 0,C 180,E1 -8373.563,E2 -8373.563} C_VEL
LIN {X 0,Y 452.546,Z 549.648,A -85,B 0,C 180,E1 -8374.901,E2 -8374.901} C_VEL
LIN {X 0,Y 452.612,Z 545.056,A -85,B 0,C 180,E1 -8376.397,E2 -8376.397} C_VEL
LIN {X 0,Y 452.842,Z 538.386,A -85,B 0,C 180,E1 -8378.03,E2 -8378.03} C_VEL
LIN {X 0,Y 453.13,Z 531.376,A -85,B 0,C 180,E1 -8379.374,E2 -8379.374} C_VEL
LIN {X 0,Y 453.543,Z 522.582,A -85,B 0,C 180,E1 -8380.718,E2 -8380.718} C_VEL
LIN {X 0,Y 454.133,Z 512.595,A -85,B 0,C 180,E1 -8381.947,E2 -8381.947} C_VEL
LIN {X 0,Y 454.642,Z 502.297,A -85,B 0,C 180,E1 -8382.965,E2 -8382.965} C_VEL
LIN {X 0,Y 455.152,Z 491.13,A -85,B 0,C 180,E1 -8383.848,E2 -8383.848} C_VEL
LIN {X 0,Y 455.732,Z 478.429,A -85,B 0,C 180,E1 -8384.628,E2 -8384.628} C_VEL
LIN {X 0,Y 456.189,Z 466.01,A -85,B 0,C 180,E1 -8385.184,E2 -8385.184} C_VEL
LIN {X 0,Y 456.652,Z 452.196,A -85,B 0,C 180,E1 -8385.597,E2 -8385.597} C_VEL
LIN {X 0,Y 457.409,Z 364.388,A -85,B 0,C 180,E1 -8387.007,E2 -8387.007} C_VEL
LIN {X 0,Y 454.263,Z 343.075,A -85,B 0,C 180,E1 -8387.467,E2 -8387.467} C_VEL
LIN {X 0,Y 454.983,Z 326.75,A -85,B 0,C 180,E1 -8390.339,E2 -8390.339} C_VEL
LIN {X 0,Y 455.883,Z 308.247,A -85,B 0,C 180,E1 -8393.631,E2 -8393.631} C_VEL
LIN {X 0,Y 455.467,Z 303.891,A -85,B 0,C 180,E1 -8394.44,E2 -8394.44} C_VEL
LIN {X 0,Y 453.551,Z 293.992,A -85,B 0,C 180,E1 -8396.377,E2 -8396.377} C_VEL
LIN {X 0,Y 453.514,Z 293.992,A -85,B 0,C 180,E1 -8398.713,E2 -8398.713} C_VEL
LIN {X 0,Y 453.469,Z 293.997,A -85,B 0,C 180,E1 -8401.8,E2 -8401.8} C_VEL
LIN {X 0,Y 453.482,Z 293.993,A -85,B 0,C 180,E1 -8404.99,E2 -8404.99} C_VEL
LIN {X 0,Y 453.465,Z 294.002,A -85,B 0,C 180,E1 -8408.313,E2 -8408.313} C_VEL
LIN {X 0,Y 453.5,Z 293.997,A -85,B 0,C 180,E1 -8410.609,E2 -8410.609} C_VEL
LIN {X 0,Y 453.459,Z 293.996,A -85,B 0,C 180,E1 -8413.244,E2 -8413.244} C_VEL
LIN {X 0,Y 453.469,Z 293.994,A -85,B 0,C 180,E1 -8415.779,E2 -8415.779} C_VEL
LIN {X 0,Y 453.485,Z 293.994,A -85,B 0,C 180,E1 -8418.21,E2 -8418.21} C_VEL
LIN {X 0,Y 453.497,Z 293.999,A -85,B 0,C 180,E1 -8420.794,E2 -8420.794} C_VEL
LIN {X 0,Y 453.46,Z 293.995,A -85,B 0,C 180,E1 -8423.917,E2 -8423.917} C_VEL
LIN {X 0,Y 453.48,Z 293.999,A -85,B 0,C 180,E1 -8427.151,E2 -8427.151} C_VEL
LIN {X 0,Y 453.481,Z 293.992,A -85,B 0,C 180,E1 -8430.268,E2 -8430.268} C_VEL
LIN {X 0,Y 453.511,Z 293.996,A -85,B 0,C 180,E1 -8433.294,E2 -8433.294} C_VEL
LIN {X 0,Y 453.508,Z 293.989,A -85,B 0,C 180,E1 -8436.239,E2 -8436.239} C_VEL
LIN {X 0,Y 453.488,Z 293.996,A -85,B 0,C 180,E1 -8439.118,E2 -8439.118} C_VEL
LIN {X 0,Y 453.509,Z 293.992,A -85,B 0,C 180,E1 -8441.944,E2 -8441.944} C_VEL
LIN {X 0,Y 453.545,Z 293.984,A -85,B 0,C 180,E1 -8444.726,E2 -8444.726} C_VEL
LIN {X 0,Y 453.564,Z 293.983,A -85,B 0,C 180,E1 -8448.379,E2 -8448.379} C_VEL
LIN {X 0,Y 453.595,Z 293.978,A -85,B 0,C 180,E1 -8451.086,E2 -8451.086} C_VEL
LIN {X 0,Y 453.655,Z 293.977,A -85,B 0,C 180,E1 -8453.774,E2 -8453.774} C_VEL
LIN {X 0,Y 453.748,Z 293.96,A -85,B 0,C 180,E1 -8457.337,E2 -8457.337} C_VEL
LIN {X 0,Y 453.826,Z 293.956,A -85,B 0,C 180,E1 -8460,E2 -8460} C_VEL
LIN {X 0,Y 453.747,Z 293.961,A -85,B 0,C 180,E1 -8462.663,E2 -8462.663} C_VEL
LIN {X 0,Y 453.67,Z 293.976,A -85,B 0,C 180,E1 -8466.225,E2 -8466.225} C_VEL
LIN {X 0,Y 453.59,Z 293.981,A -85,B 0,C 180,E1 -8468.913,E2 -8468.913} C_VEL
LIN {X 0,Y 453.569,Z 293.99,A -85,B 0,C 180,E1 -8472.529,E2 -8472.529} C_VEL
LIN {X 0,Y 453.55,Z 293.986,A -85,B 0,C 180,E1 -8476.196,E2 -8476.196} C_VEL
LIN {X 0,Y 453.522,Z 293.991,A -85,B 0,C 180,E1 -8479.039,E2 -8479.039} C_VEL
LIN {X 0,Y 453.481,Z 293.992,A -85,B 0,C 180,E1 -8481.836,E2 -8481.836} C_VEL
LIN {X 0,Y 453.518,Z 293.993,A -85,B 0,C 180,E1 -8484.734,E2 -8484.734} C_VEL
LIN {X 0,Y 453.537,Z 293.985,A -85,B 0,C 180,E1 -8487.959,E2 -8487.959} C_VEL
LIN {X 0,Y 453.47,Z 293.997,A -85,B 0,C 180,E1 -8491.524,E2 -8491.524} C_VEL
LIN {X 0,Y 453.491,Z 293.993,A -85,B 0,C 180,E1 -8494.777,E2 -8494.777} C_VEL
LIN {X 0,Y 453.467,Z 293.994,A -85,B 0,C 180,E1 -8498.311,E2 -8498.311} C_VEL
LIN {X 0,Y 453.498,Z 293.99,A -85,B 0,C 180,E1 -8500.608,E2 -8500.608} C_VEL
LIN {X 0,Y 453.459,Z 294,A -85,B 0,C 180,E1 -8503.243,E2 -8503.243} C_VEL
LIN {X 0,Y 453.466,Z 294,A -85,B 0,C 180,E1 -8505.778,E2 -8505.778} C_VEL
LIN {X 0,Y 453.483,Z 293.994,A -85,B 0,C 180,E1 -8508.209,E2 -8508.209} C_VEL
LIN {X 0,Y 453.491,Z 293.991,A -85,B 0,C 180,E1 -8510.794,E2 -8510.794} C_VEL
LIN {X 0,Y 453.458,Z 294.003,A -85,B 0,C 180,E1 -8513.916,E2 -8513.916} C_VEL
LIN {X 0,Y 453.486,Z 293.992,A -85,B 0,C 180,E1 -8517.15,E2 -8517.15} C_VEL
LIN {X 0,Y 453.479,Z 293.998,A -85,B 0,C 180,E1 -8520.267,E2 -8520.267} C_VEL
LIN {X 0,Y 453.505,Z 293.989,A -85,B 0,C 180,E1 -8523.293,E2 -8523.293} C_VEL
LIN {X 0,Y 453.501,Z 293.998,A -85,B 0,C 180,E1 -8526.238,E2 -8526.238} C_VEL
LIN {X 0,Y 453.485,Z 293.992,A -85,B 0,C 180,E1 -8529.117,E2 -8529.117} C_VEL
LIN {X 0,Y 453.513,Z 293.99,A -85,B 0,C 180,E1 -8531.943,E2 -8531.943} C_VEL
LIN {X 0,Y 453.542,Z 293.991,A -85,B 0,C 180,E1 -8534.725,E2 -8534.725} C_VEL
LIN {X 0,Y 453.561,Z 293.987,A -85,B 0,C 180,E1 -8538.378,E2 -8538.378} C_VEL
LIN {X 0,Y 453.587,Z 293.986,A -85,B 0,C 180,E1 -8541.085,E2 -8541.085} C_VEL
LIN {X 0,Y 453.619,Z 293.983,A -85,B 0,C 180,E1 -8543.079,E2 -8543.079} C_VEL
LIN {X 0,Y 453.352,Z 294.423,A -85,B 0,C 180,E1 -8543.569,E2 -8543.569} C_VEL
LIN {X 0,Y 452.663,Z 295.565,A -85,B 0,C 180,E1 -8544.037,E2 -8544.037} C_VEL
LIN {X 0,Y 450.63,Z 299.139,A -85,B 0,C 180,E1 -8544.908,E2 -8544.908} C_VEL
LIN {X 0,Y 448.557,Z 303.624,A -85,B 0,C 180,E1 -8545.749,E2 -8545.749} C_VEL
LIN {X 0,Y 447.668,Z 306.911,A -85,B 0,C 180,E1 -8546.392,E2 -8546.392} C_VEL
LIN {X 0,Y 447.598,Z 307.98,A -85,B 0,C 180,E1 -8546.611,E2 -8546.611} C_VEL
LIN {X 0,Y 447.538,Z 311.575,A -85,B 0,C 180,E1 -8547.354,E2 -8547.354} C_VEL
LIN {X 0,Y 450.828,Z 329.522,A -85,B 0,C 180,E1 -8547.782,E2 -8547.782} C_VEL
LIN {X 0,Y 449.875,Z 419.13,A -85,B 0,C 180,E1 -8549.235,E2 -8549.235} C_VEL
LIN {X 0,Y 449.537,Z 432.412,A -85,B 0,C 180,E1 -8549.634,E2 -8549.634} C_VEL
LIN {X 0,Y 449.222,Z 445.412,A -85,B 0,C 180,E1 -8550.223,E2 -8550.223} C_VEL
LIN {X 0,Y 448.744,Z 456.454,A -85,B 0,C 180,E1 -8550.896,E2 -8550.896} C_VEL
LIN {X 0,Y 448.124,Z 467.971,A -85,B 0,C 180,E1 -8551.796,E2 -8551.796} C_VEL
LIN {X 0,Y 447.509,Z 478.347,A -85,B 0,C 180,E1 -8552.812,E2 -8552.812} C_VEL
LIN {X 0,Y 447.059,Z 486.817,A -85,B 0,C 180,E1 -8553.83,E2 -8553.83} C_VEL
LIN {X 0,Y 446.634,Z 494.635,A -85,B 0,C 180,E1 -8554.963,E2 -8554.963} C_VEL
LIN {X 0,Y 446.238,Z 502.276,A -85,B 0,C 180,E1 -8556.328,E2 -8556.328} C_VEL
LIN {X 0,Y 445.964,Z 508.423,A -85,B 0,C 180,E1 -8557.697,E2 -8557.697} C_VEL
LIN {X 0,Y 445.675,Z 513.321,A -85,B 0,C 180,E1 -8559.072,E2 -8559.072} C_VEL
LIN {X 0,Y 445.579,Z 517.08,A -85,B 0,C 180,E1 -8560.449,E2 -8560.449} C_VEL
LIN {X 0,Y 445.427,Z 520.042,A -85,B 0,C 180,E1 -8561.974,E2 -8561.974} C_VEL
LIN {X 0,Y 445.291,Z 521.984,A -85,B 0,C 180,E1 -8563.693,E2 -8563.693} C_VEL
LIN {X 0,Y 445.3,Z 522.401,A -85,B 0,C 180,E1 -8564.625,E2 -8564.625} C_VEL
LIN {X 0,Y 445.321,Z 522.395,A -85,B 0,C 180,E1 -8565.7,E2 -8565.7} C_VEL
LIN {X 0,Y 445.298,Z 521.19,A -85,B 0,C 180,E1 -8567.448,E2 -8567.448} C_VEL
LIN {X 0,Y 445.453,Z 519.23,A -85,B 0,C 180,E1 -8568.803,E2 -8568.803} C_VEL
LIN {X 0,Y 445.611,Z 515.944,A -85,B 0,C 180,E1 -8570.301,E2 -8570.301} C_VEL
LIN {X 0,Y 445.861,Z 511.297,A -85,B 0,C 180,E1 -8571.828,E2 -8571.828} C_VEL
LIN {X 0,Y 446.152,Z 505.932,A -85,B 0,C 180,E1 -8573.19,E2 -8573.19} C_VEL
LIN {X 0,Y 446.588,Z 498.727,A -85,B 0,C 180,E1 -8574.646,E2 -8574.646} C_VEL
LIN {X 0,Y 447.058,Z 491.244,A -85,B 0,C 180,E1 -8575.863,E2 -8575.863} C_VEL
LIN {X 0,Y 447.651,Z 482.007,A -85,B 0,C 180,E1 -8577.082,E2 -8577.082} C_VEL
LIN {X 0,Y 448.298,Z 471.194,A -85,B 0,C 180,E1 -8578.233,E2 -8578.233} C_VEL
LIN {X 0,Y 448.948,Z 460.243,A -85,B 0,C 180,E1 -8579.158,E2 -8579.158} C_VEL
LIN {X 0,Y 449.528,Z 448.141,A -85,B 0,C 180,E1 -8579.953,E2 -8579.953} C_VEL
LIN {X 0,Y 450.034,Z 435.59,A -85,B 0,C 180,E1 -8580.571,E2 -8580.571} C_VEL
LIN {X 0,Y 450.332,Z 422.502,A -85,B 0,C 180,E1 -8581.012,E2 -8581.012} C_VEL
LIN {X 0,Y 450.672,Z 403.804,A -85,B 0,C 180,E1 -8581.362,E2 -8581.362} C_VEL
LIN {X 0,Y 451.413,Z 328.724,A -85,B 0,C 180,E1 -8582.578,E2 -8582.578} C_VEL
LIN {X 0,Y 447.824,Z 311.579,A -85,B 0,C 180,E1 -8583.042,E2 -8583.042} C_VEL
LIN {X 0,Y 447.864,Z 302.27,A -85,B 0,C 180,E1 -8584.932,E2 -8584.932} C_VEL
LIN {X 0,Y 446.382,Z 294.884,A -85,B 0,C 180,E1 -8586.586,E2 -8586.586} C_VEL
LIN {X 0,Y 446.383,Z 294.884,A -85,B 0,C 180,E1 -8589.514,E2 -8589.514} C_VEL
LIN {X 0,Y 446.36,Z 294.884,A -85,B 0,C 180,E1 -8592.61,E2 -8592.61} C_VEL
LIN {X 0,Y 446.437,Z 294.877,A -85,B 0,C 180,E1 -8595.103,E2 -8595.103} C_VEL
LIN {X 0,Y 446.393,Z 294.878,A -85,B 0,C 180,E1 -8598.605,E2 -8598.605} C_VEL
LIN {X 0,Y 446.386,Z 294.883,A -85,B 0,C 180,E1 -8601.923,E2 -8601.923} C_VEL
LIN {X 0,Y 446.408,Z 294.871,A -85,B 0,C 180,E1 -8605.475,E2 -8605.475} C_VEL
LIN {X 0,Y 446.401,Z 294.873,A -85,B 0,C 180,E1 -8608.699,E2 -8608.699} C_VEL
LIN {X 0,Y 446.436,Z 294.874,A -85,B 0,C 180,E1 -8611.829,E2 -8611.829} C_VEL
LIN {X 0,Y 446.424,Z 294.87,A -85,B 0,C 180,E1 -8614.846,E2 -8614.846} C_VEL
LIN {X 0,Y 446.434,Z 294.871,A -85,B 0,C 180,E1 -8618.245,E2 -8618.245} C_VEL
LIN {X 0,Y 446.436,Z 294.874,A -85,B 0,C 180,E1 -8621.648,E2 -8621.648} C_VEL
LIN {X 0,Y 446.491,Z 294.867,A -85,B 0,C 180,E1 -8624.479,E2 -8624.479} C_VEL
LIN {X 0,Y 446.502,Z 294.863,A -85,B 0,C 180,E1 -8628.193,E2 -8628.193} C_VEL
LIN {X 0,Y 446.523,Z 294.861,A -85,B 0,C 180,E1 -8630.945,E2 -8630.945} C_VEL
LIN {X 0,Y 446.603,Z 294.845,A -85,B 0,C 180,E1 -8633.676,E2 -8633.676} C_VEL
LIN {X 0,Y 446.676,Z 294.837,A -85,B 0,C 180,E1 -8637.295,E2 -8637.295} C_VEL
LIN {X 0,Y 446.777,Z 294.828,A -85,B 0,C 180,E1 -8640,E2 -8640} C_VEL
LIN {X 0,Y 446.677,Z 294.839,A -85,B 0,C 180,E1 -8642.706,E2 -8642.706} C_VEL
LIN {X 0,Y 446.625,Z 294.85,A -85,B 0,C 180,E1 -8646.324,E2 -8646.324} C_VEL
LIN {X 0,Y 446.525,Z 294.861,A -85,B 0,C 180,E1 -8649.056,E2 -8649.056} C_VEL
LIN {X 0,Y 446.507,Z 294.864,A -85,B 0,C 180,E1 -8652.73,E2 -8652.73} C_VEL
LIN {X 0,Y 446.483,Z 294.866,A -85,B 0,C 180,E1 -8656.229,E2 -8656.229} C_VEL
LIN {X 0,Y 446.456,Z 294.87,A -85,B 0,C 180,E1 -8659.304,E2 -8659.304} C_VEL
LIN {X 0,Y 446.405,Z 294.875,A -85,B 0,C 180,E1 -8662.2,E2 -8662.2} C_VEL
LIN {X 0,Y 446.447,Z 294.875,A -85,B 0,C 180,E1 -8665.153,E2 -8665.153} C_VEL
LIN {X 0,Y 446.473,Z 294.861,A -85,B 0,C 180,E1 -8668.18,E2 -8668.18} C_VEL
LIN {X 0,Y 446.423,Z 294.876,A -85,B 0,C 180,E1 -8671.3,E2 -8671.3} C_VEL
LIN {X 0,Y 446.42,Z 294.875,A -85,B 0,C 180,E1 -8674.524,E2 -8674.524} C_VEL
LIN {X 0,Y 446.429,Z 294.874,A -85,B 0,C 180,E1 -8678.084,E2 -8678.084} C_VEL
LIN {X 0,Y 446.435,Z 294.875,A -85,B 0,C 180,E1 -8680.922,E2 -8680.922} C_VEL
LIN {X 0,Y 446.414,Z 294.877,A -85,B 0,C 180,E1 -8683.845,E2 -8683.845} C_VEL
LIN {X 0,Y 446.439,Z 294.867,A -85,B 0,C 180,E1 -8686.398,E2 -8686.398} C_VEL
LIN {X 0,Y 446.461,Z 294.868,A -85,B 0,C 180,E1 -8689.806,E2 -8689.806} C_VEL
LIN {X 0,Y 446.426,Z 294.877,A -85,B 0,C 180,E1 -8692.125,E2 -8692.125} C_VEL
LIN {X 0,Y 446.425,Z 294.879,A -85,B 0,C 180,E1 -8695.479,E2 -8695.479} C_VEL
LIN {X 0,Y 446.411,Z 294.875,A -85,B 0,C 180,E1 -8698.701,E2 -8698.701} C_VEL
LIN {X 0,Y 446.481,Z 294.871,A -85,B 0,C 180,E1 -8701.823,E2 -8701.823} C_VEL
LIN {X 0,Y 446.539,Z 295.006,A -85,B 0,C 180,E1 -8703.075,E2 -8703.075} C_VEL
LIN {X 0,Y 449.038,Z 307.686,A -85,B 0,C 180,E1 -8705.649,E2 -8705.649} C_VEL
LIN {X 0,Y 449.088,Z 313.416,A -85,B 0,C 180,E1 -8706.726,E2 -8706.726} C_VEL
LIN {X 0,Y 448.097,Z 330.377,A -85,B 0,C 180,E1 -8709.817,E2 -8709.817} C_VEL
LIN {X 0,Y 447.521,Z 342.551,A -85,B 0,C 180,E1 -8712.002,E2 -8712.002} C_VEL
LIN {X 0,Y 451.063,Z 364.83,A -85,B 0,C 180,E1 -8712.534,E2 -8712.534} C_VEL
LIN {X 0,Y 450.268,Z 450.842,A -85,B 0,C 180,E1 -8713.946,E2 -8713.946} C_VEL
LIN {X 0,Y 449.824,Z 464.11,A -85,B 0,C 180,E1 -8714.337,E2 -8714.337} C_VEL
LIN {X 0,Y 449.295,Z 476.269,A -85,B 0,C 180,E1 -8714.87,E2 -8714.87} C_VEL
LIN {X 0,Y 448.649,Z 488.564,A -85,B 0,C 180,E1 -8715.602,E2 -8715.602} C_VEL
LIN {X 0,Y 447.994,Z 500.255,A -85,B 0,C 180,E1 -8716.515,E2 -8716.515} C_VEL
LIN {X 0,Y 447.425,Z 510.621,A -85,B 0,C 180,E1 -8717.528,E2 -8717.528} C_VEL
LIN {X 0,Y 446.838,Z 520.06,A -85,B 0,C 180,E1 -8718.663,E2 -8718.663} C_VEL
LIN {X 0,Y 446.25,Z 529.175,A -85,B 0,C 180,E1 -8720.025,E2 -8720.025} C_VEL
LIN {X 0,Y 445.883,Z 536.539,A -85,B 0,C 180,E1 -8721.39,E2 -8721.39} C_VEL
LIN {X 0,Y 445.635,Z 542.456,A -85,B 0,C 180,E1 -8722.753,E2 -8722.753} C_VEL
LIN {X 0,Y 445.469,Z 546.628,A -85,B 0,C 180,E1 -8723.957,E2 -8723.957} C_VEL
LIN {X 0,Y 445.412,Z 550.697,A -85,B 0,C 180,E1 -8725.476,E2 -8725.476} C_VEL
LIN {X 0,Y 445.38,Z 552.522,A -85,B 0,C 180,E1 -8726.383,E2 -8726.383} C_VEL
LIN {X 0,Y 445.432,Z 553.9,A -85,B 0,C 180,E1 -8727.288,E2 -8727.288} C_VEL
LIN {X 0,Y 445.341,Z 555.471,A -85,B 0,C 180,E1 -8729.097,E2 -8729.097} C_VEL
LIN {X 0,Y 445.371,Z 555.653,A -85,B 0,C 180,E1 -8730.001,E2 -8730.001} C_VEL
LIN {X 0,Y 445.375,Z 554.781,A -85,B 0,C 180,E1 -8731.81,E2 -8731.81} C_VEL
LIN {X 0,Y 445.433,Z 553.763,A -85,B 0,C 180,E1 -8732.714,E2 -8732.714} C_VEL
LIN {X 0,Y 445.384,Z 552.316,A -85,B 0,C 180,E1 -8733.62,E2 -8733.62} C_VEL
LIN {X 0,Y 445.474,Z 549.326,A -85,B 0,C 180,E1 -8734.979,E2 -8734.979} C_VEL
LIN {X 0,Y 445.557,Z 543.812,A -85,B 0,C 180,E1 -8736.75,E2 -8736.75} C_VEL
LIN {X 0,Y 445.77,Z 538.02,A -85,B 0,C 180,E1 -8738.159,E2 -8738.159} C_VEL
LIN {X 0,Y 446.073,Z 530.978,A -85,B 0,C 180,E1 -8739.523,E2 -8739.523} C_VEL
LIN {X 0,Y 446.536,Z 522.153,A -85,B 0,C 180,E1 -8740.888,E2 -8740.888} C_VEL
LIN {X 0,Y 447.156,Z 512.132,A -85,B 0,C 180,E1 -8742.136,E2 -8742.136} C_VEL
LIN {X 0,Y 447.657,Z 501.767,A -85,B 0,C 180,E1 -8743.171,E2 -8743.171} C_VEL
LIN {X 0,Y 448.199,Z 490.54,A -85,B 0,C 180,E1 -8744.068,E2 -8744.068} C_VEL
LIN {X 0,Y 448.799,Z 478.761,A -85,B 0,C 180,E1 -8744.801,E2 -8744.801} C_VEL
LIN {X 0,Y 449.291,Z 465.861,A -85,B 0,C 180,E1 -8745.394,E2 -8745.394} C_VEL
LIN {X 0,Y 449.778,Z 452.089,A -85,B 0,C 180,E1 -8745.812,E2 -8745.812} C_VEL
LIN {X 0,Y 450.519,Z 364.449,A -85,B 0,C 180,E1 -8747.242,E2 -8747.242} C_VEL
LIN {X 0,Y 447.291,Z 342.71,A -85,B 0,C 180,E1 -8747.737,E2 -8747.737} C_VEL
LIN {X 0,Y 448.136,Z 325.003,A -85,B 0,C 180,E1 -8750.904,E2 -8750.904} C_VEL
LIN {X 0,Y 448.914,Z 309.114,A -85,B 0,C 180,E1 -8753.775,E2 -8753.775} C_VEL
LIN {X 0,Y 448.039,Z 302.384,A -85,B 0,C 180,E1 -8755.059,E2 -8755.059} C_VEL
LIN {X 0,Y 446.518,Z 294.867,A -85,B 0,C 180,E1 -8756.562,E2 -8756.562} C_VEL
LIN {X 0,Y 446.453,Z 294.871,A -85,B 0,C 180,E1 -8759.21,E2 -8759.21} C_VEL
LIN {X 0,Y 446.426,Z 294.877,A -85,B 0,C 180,E1 -8762.362,E2 -8762.362} C_VEL
LIN {X 0,Y 446.424,Z 294.872,A -85,B 0,C 180,E1 -8765.627,E2 -8765.627} C_VEL
LIN {X 0,Y 446.431,Z 294.872,A -85,B 0,C 180,E1 -8769.03,E2 -8769.03} C_VEL
LIN {X 0,Y 446.44,Z 294.874,A -85,B 0,C 180,E1 -8772.278,E2 -8772.278} C_VEL
LIN {X 0,Y 446.457,Z 294.87,A -85,B 0,C 180,E1 -8775.104,E2 -8775.104} C_VEL
LIN {X 0,Y 446.434,Z 294.877,A -85,B 0,C 180,E1 -8778.609,E2 -8778.609} C_VEL
LIN {X 0,Y 446.447,Z 294.875,A -85,B 0,C 180,E1 -8780.973,E2 -8780.973} C_VEL
LIN {X 0,Y 446.423,Z 294.873,A -85,B 0,C 180,E1 -8784.374,E2 -8784.374} C_VEL
LIN {X 0,Y 446.422,Z 294.873,A -85,B 0,C 180,E1 -8787.638,E2 -8787.638} C_VEL
LIN {X 0,Y 446.454,Z 294.871,A -85,B 0,C 180,E1 -8790.791,E2 -8790.791} C_VEL
LIN {X 0,Y 446.484,Z 294.865,A -85,B 0,C 180,E1 -8793.849,E2 -8793.849} C_VEL
LIN {X 0,Y 446.434,Z 294.872,A -85,B 0,C 180,E1 -8796.823,E2 -8796.823} C_VEL
LIN {X 0,Y 446.45,Z 294.872,A -85,B 0,C 180,E1 -8799.737,E2 -8799.737} C_VEL
LIN {X 0,Y 446.462,Z 294.866,A -85,B 0,C 180,E1 -8802.597,E2 -8802.597} C_VEL
LIN {X 0,Y 446.475,Z 294.87,A -85,B 0,C 180,E1 -8805.412,E2 -8805.412} C_VEL
LIN {X 0,Y 446.523,Z 294.861,A -85,B 0,C 180,E1 -8808.193,E2 -8808.193} C_VEL
LIN {X 0,Y 446.541,Z 294.857,A -85,B 0,C 180,E1 -8810.945,E2 -8810.945} C_VEL
LIN {X 0,Y 446.624,Z 294.852,A -85,B 0,C 180,E1 -8813.676,E2 -8813.676} C_VEL
LIN {X 0,Y 446.695,Z 294.838,A -85,B 0,C 180,E1 -8817.294,E2 -8817.294} C_VEL
LIN {X 0,Y 446.796,Z 294.832,A -85,B 0,C 180,E1 -8820,E2 -8820} C_VEL
LIN {X 0,Y 446.694,Z 294.84,A -85,B 0,C 180,E1 -8822.705,E2 -8822.705} C_VEL
LIN {X 0,Y 446.639,Z 294.853,A -85,B 0,C 180,E1 -8826.324,E2 -8826.324} C_VEL
LIN {X 0,Y 446.537,Z 294.858,A -85,B 0,C 180,E1 -8829.055,E2 -8829.055} C_VEL
LIN {X 0,Y 446.527,Z 294.864,A -85,B 0,C 180,E1 -8832.729,E2 -8832.729} C_VEL
LIN {X 0,Y 446.501,Z 294.865,A -85,B 0,C 180,E1 -8836.227,E2 -8836.227} C_VEL
LIN {X 0,Y 446.473,Z 294.867,A -85,B 0,C 180,E1 -8839.303,E2 -8839.303} C_VEL
LIN {X 0,Y 446.423,Z 294.873,A -85,B 0,C 180,E1 -8842.199,E2 -8842.199} C_VEL
LIN {X 0,Y 446.463,Z 294.872,A -85,B 0,C 180,E1 -8845.152,E2 -8845.152} C_VEL
LIN {X 0,Y 446.49,Z 294.863,A -85,B 0,C 180,E1 -8848.178,E2 -8848.178} C_VEL
LIN {X 0,Y 446.423,Z 294.873,A -85,B 0,C 180,E1 -8851.774,E2 -8851.774} C_VEL
LIN {X 0,Y 446.432,Z 294.871,A -85,B 0,C 180,E1 -8854.523,E2 -8854.523} C_VEL
LIN {X 0,Y 446.418,Z 294.873,A -85,B 0,C 180,E1 -8858.078,E2 -8858.078} C_VEL
LIN {X 0,Y 446.431,Z 294.872,A -85,B 0,C 180,E1 -8860.917,E2 -8860.917} C_VEL
LIN {X 0,Y 446.404,Z 294.878,A -85,B 0,C 180,E1 -8863.845,E2 -8863.845} C_VEL
LIN {X 0,Y 446.4,Z 294.875,A -85,B 0,C 180,E1 -8866.403,E2 -8866.403} C_VEL
LIN {X 0,Y 446.43,Z 294.872,A -85,B 0,C 180,E1 -8869.082,E2 -8869.082} C_VEL
LIN {X 0,Y 446.411,Z 294.877,A -85,B 0,C 180,E1 -8872.12,E2 -8872.12} C_VEL
LIN {X 0,Y 446.433,Z 294.873,A -85,B 0,C 180,E1 -8875.476,E2 -8875.476} C_VEL
LIN {X 0,Y 446.419,Z 294.873,A -85,B 0,C 180,E1 -8878.699,E2 -8878.699} C_VEL
LIN {X 0,Y 446.488,Z 294.867,A -85,B 0,C 180,E1 -8881.82,E2 -8881.82} C_VEL
LIN {X 0,Y 446.447,Z 294.87,A -85,B 0,C 180,E1 -8884.846,E2 -8884.846} C_VEL
LIN {X 0,Y 446.451,Z 294.875,A -85,B 0,C 180,E1 -8888.244,E2 -8888.244} C_VEL
LIN {X 0,Y 446.459,Z 294.867,A -85,B 0,C 180,E1 -8891.648,E2 -8891.648} C_VEL
LIN {X 0,Y 446.51,Z 294.868,A -85,B 0,C 180,E1 -8894.479,E2 -8894.479} C_VEL
LIN {X 0,Y 446.519,Z 294.862,A -85,B 0,C 180,E1 -8898.192,E2 -8898.192} C_VEL
LIN {X 0,Y 446.534,Z 294.866,A -85,B 0,C 180,E1 -8900.943,E2 -8900.943} C_VEL
LIN {X 0,Y 446.638,Z 294.992,A -85,B 0,C 180,E1 -8903.845,E2 -8903.845} C_VEL
LIN {X 0,Y 447.781,Z 302.588,A -85,B 0,C 180,E1 -8905.498,E2 -8905.498} C_VEL
LIN {X 0,Y 447.598,Z 307.98,A -85,B 0,C 180,E1 -8906.611,E2 -8906.611} C_VEL
LIN {X 0,Y 447.149,Z 310.181,A -85,B 0,C 180,E1 -8906.917,E2 -8906.917} C_VEL
LIN {X 0,Y 445.802,Z 313.776,A -85,B 0,C 180,E1 -8907.165,E2 -8907.165} C_VEL
LIN {X 0,Y 443.807,Z 319.334,A -85,B 0,C 180,E1 -8907.337,E2 -8907.337} C_VEL
LIN {X 0,Y 443.189,Z 323.388,A -85,B 0,C 180,E1 -8907.402,E2 -8907.402} C_VEL
LIN {X 0,Y 443.914,Z 338.275,A -85,B 0,C 180,E1 -8907.678,E2 -8907.678} C_VEL
LIN {X 0,Y 443.017,Z 419.005,A -85,B 0,C 180,E1 -8909.005,E2 -8909.005} C_VEL
LIN {X 0,Y 442.656,Z 432.174,A -85,B 0,C 180,E1 -8909.401,E2 -8909.401} C_VEL
LIN {X 0,Y 442.315,Z 445.323,A -85,B 0,C 180,E1 -8909.999,E2 -8909.999} C_VEL
LIN {X 0,Y 441.838,Z 456.45,A -85,B 0,C 180,E1 -8910.682,E2 -8910.682} C_VEL
LIN {X 0,Y 441.184,Z 468.019,A -85,B 0,C 180,E1 -8911.596,E2 -8911.596} C_VEL
LIN {X 0,Y 440.532,Z 478.435,A -85,B 0,C 180,E1 -8912.627,E2 -8912.627} C_VEL
LIN {X 0,Y 440.064,Z 486.933,A -85,B 0,C 180,E1 -8913.661,E2 -8913.661} C_VEL
LIN {X 0,Y 439.608,Z 494.785,A -85,B 0,C 180,E1 -8914.813,E2 -8914.813} C_VEL
LIN {X 0,Y 439.179,Z 502.46,A -85,B 0,C 180,E1 -8916.2,E2 -8916.2} C_VEL
LIN {X 0,Y 438.963,Z 507.711,A -85,B 0,C 180,E1 -8917.357,E2 -8917.357} C_VEL
LIN {X 0,Y 438.669,Z 512.814,A -85,B 0,C 180,E1 -8918.753,E2 -8918.753} C_VEL
LIN {X 0,Y 438.487,Z 516.773,A -85,B 0,C 180,E1 -8920.153,E2 -8920.153} C_VEL
LIN {X 0,Y 438.406,Z 518.81,A -85,B 0,C 180,E1 -8921.09,E2 -8921.09} C_VEL
LIN {X 0,Y 438.332,Z 520.43,A -85,B 0,C 180,E1 -8922.029,E2 -8922.029} C_VEL
LIN {X 0,Y 438.249,Z 521.628,A -85,B 0,C 180,E1 -8922.973,E2 -8922.973} C_VEL
LIN {X 0,Y 438.189,Z 522.368,A -85,B 0,C 180,E1 -8923.919,E2 -8923.919} C_VEL
LIN {X 0,Y 438.23,Z 522.706,A -85,B 0,C 180,E1 -8924.867,E2 -8924.867} C_VEL
LIN {X 0,Y 438.235,Z 522.647,A -85,B 0,C 180,E1 -8925.819,E2 -8925.819} C_VEL
LIN {X 0,Y 438.193,Z 522.135,A -85,B 0,C 180,E1 -8926.778,E2 -8926.778} C_VEL
LIN {X 0,Y 438.237,Z 521.185,A -85,B 0,C 180,E1 -8927.739,E2 -8927.739} C_VEL
LIN {X 0,Y 438.4,Z 519.392,A -85,B 0,C 180,E1 -8928.946,E2 -8928.946} C_VEL
LIN {X 0,Y 438.574,Z 515.607,A -85,B 0,C 180,E1 -8930.641,E2 -8930.641} C_VEL
LIN {X 0,Y 438.84,Z 511.086,A -85,B 0,C 180,E1 -8932.106,E2 -8932.106} C_VEL
LIN {X 0,Y 439.211,Z 505.216,A -85,B 0,C 180,E1 -8933.579,E2 -8933.579} C_VEL
LIN {X 0,Y 439.701,Z 497.701,A -85,B 0,C 180,E1 -8935.058,E2 -8935.058} C_VEL
LIN {X 0,Y 440.251,Z 489.921,A -85,B 0,C 180,E1 -8936.293,E2 -8936.293} C_VEL
LIN {X 0,Y 440.874,Z 480.348,A -85,B 0,C 180,E1 -8937.533,E2 -8937.533} C_VEL
LIN {X 0,Y 441.554,Z 469.531,A -85,B 0,C 180,E1 -8938.653,E2 -8938.653} C_VEL
LIN {X 0,Y 442.293,Z 457.375,A -85,B 0,C 180,E1 -8939.64,E2 -8939.64} C_VEL
LIN {X 0,Y 442.864,Z 445.469,A -85,B 0,C 180,E1 -8940.385,E2 -8940.385} C_VEL
LIN {X 0,Y 443.387,Z 432.24,A -85,B 0,C 180,E1 -8940.985,E2 -8940.985} C_VEL
LIN {X 0,Y 443.686,Z 419.566,A -85,B 0,C 180,E1 -8941.373,E2 -8941.373} C_VEL
LIN {X 0,Y 444.741,Z 329.745,A -85,B 0,C 180,E1 -8942.871,E2 -8942.871} C_VEL
LIN {X 0,Y 441.14,Z 312.935,A -85,B 0,C 180,E1 -8943.334,E2 -8943.334} C_VEL
LIN {X 0,Y 440.911,Z 311.736,A -85,B 0,C 180,E1 -8943.392,E2 -8943.392} C_VEL
LIN {X 0,Y 440.97,Z 303.877,A -85,B 0,C 180,E1 -8945.01,E2 -8945.01} C_VEL
LIN {X 0,Y 439.341,Z 295.762,A -85,B 0,C 180,E1 -8946.843,E2 -8946.843} C_VEL
LIN {X 0,Y 439.335,Z 295.761,A -85,B 0,C 180,E1 -8949.839,E2 -8949.839} C_VEL
LIN {X 0,Y 439.318,Z 295.762,A -85,B 0,C 180,E1 -8952.618,E2 -8952.618} C_VEL
LIN {X 0,Y 439.385,Z 295.754,A -85,B 0,C 180,E1 -8955.269,E2 -8955.269} C_VEL
LIN {X 0,Y 439.343,Z 295.758,A -85,B 0,C 180,E1 -8959.015,E2 -8959.015} C_VEL
LIN {X 0,Y 439.324,Z 295.759,A -85,B 0,C 180,E1 -8962.563,E2 -8962.563} C_VEL
LIN {X 0,Y 439.38,Z 295.74,A -85,B 0,C 180,E1 -8964.842,E2 -8964.842} C_VEL
LIN {X 0,Y 439.358,Z 295.753,A -85,B 0,C 180,E1 -8968.139,E2 -8968.139} C_VEL
LIN {X 0,Y 439.395,Z 295.752,A -85,B 0,C 180,E1 -8971.603,E2 -8971.603} C_VEL
LIN {X 0,Y 439.362,Z 295.752,A -85,B 0,C 180,E1 -8974.413,E2 -8974.413} C_VEL
LIN {X 0,Y 439.349,Z 295.756,A -85,B 0,C 180,E1 -8977.424,E2 -8977.424} C_VEL
LIN {X 0,Y 439.426,Z 295.746,A -85,B 0,C 180,E1 -8980.663,E2 -8980.663} C_VEL
LIN {X 0,Y 439.446,Z 295.744,A -85,B 0,C 180,E1 -8984.224,E2 -8984.224} C_VEL
LIN {X 0,Y 439.469,Z 295.739,A -85,B 0,C 180,E1 -8988.001,E2 -8988.001} C_VEL
LIN {X 0,Y 439.518,Z 295.734,A -85,B 0,C 180,E1 -8991.726,E2 -8991.726} C_VEL
LIN {X 0,Y 439.593,Z 295.728,A -85,B 0,C 180,E1 -8994.496,E2 -8994.496} C_VEL
LIN {X 0,Y 439.62,Z 295.718,A -85,B 0,C 180,E1 -8998.168,E2 -8998.168} C_VEL
LIN {X 0,Y 439.747,Z 295.704,A -85,B 0,C 180,E1 -9000,E2 -9000} C_VEL
LIN {X 0,Y 439.626,Z 295.716,A -85,B 0,C 180,E1 -9002.749,E2 -9002.749} C_VEL
LIN {X 0,Y 439.599,Z 295.727,A -85,B 0,C 180,E1 -9006.426,E2 -9006.426} C_VEL
LIN {X 0,Y 439.487,Z 295.736,A -85,B 0,C 180,E1 -9009.202,E2 -9009.202} C_VEL
LIN {X 0,Y 439.451,Z 295.739,A -85,B 0,C 180,E1 -9012.938,E2 -9012.938} C_VEL
LIN {X 0,Y 439.434,Z 295.745,A -85,B 0,C 180,E1 -9016.349,E2 -9016.349} C_VEL
LIN {X 0,Y 439.389,Z 295.748,A -85,B 0,C 180,E1 -9019.627,E2 -9019.627} C_VEL
LIN {X 0,Y 439.352,Z 295.755,A -85,B 0,C 180,E1 -9022.576,E2 -9022.576} C_VEL
LIN {X 0,Y 439.394,Z 295.751,A -85,B 0,C 180,E1 -9025.586,E2 -9025.586} C_VEL
LIN {X 0,Y 439.414,Z 295.743,A -85,B 0,C 180,E1 -9028.674,E2 -9028.674} C_VEL
LIN {X 0,Y 439.374,Z 295.748,A -85,B 0,C 180,E1 -9032.035,E2 -9032.035} C_VEL
LIN {X 0,Y 439.386,Z 295.754,A -85,B 0,C 180,E1 -9035.342,E2 -9035.342} C_VEL
LIN {X 0,Y 439.389,Z 295.75,A -85,B 0,C 180,E1 -9038.595,E2 -9038.595} C_VEL
LIN {X 0,Y 439.39,Z 295.756,A -85,B 0,C 180,E1 -9041.26,E2 -9041.26} C_VEL
LIN {X 0,Y 439.398,Z 295.747,A -85,B 0,C 180,E1 -9044.73,E2 -9044.73} C_VEL
LIN {X 0,Y 439.405,Z 295.754,A -85,B 0,C 180,E1 -9047.799,E2 -9047.799} C_VEL
LIN {X 0,Y 439.442,Z 295.741,A -85,B 0,C 180,E1 -9050.231,E2 -9050.231} C_VEL
LIN {X 0,Y 439.371,Z 295.753,A -85,B 0,C 180,E1 -9053.715,E2 -9053.715} C_VEL
LIN {X 0,Y 439.367,Z 295.753,A -85,B 0,C 180,E1 -9057.056,E2 -9057.056} C_VEL
LIN {X 0,Y 439.378,Z 295.754,A -85,B 0,C 180,E1 -9060.276,E2 -9060.276} C_VEL
LIN {X 0,Y 439.476,Z 295.769,A -85,B 0,C 180,E1 -9062.759,E2 -9062.759} C_VEL
LIN {X 0,Y 441.734,Z 306.903,A -85,B 0,C 180,E1 -9065.077,E2 -9065.077} C_VEL
LIN {X 0,Y 442.312,Z 312.055,A -85,B 0,C 180,E1 -9066.1,E2 -9066.1} C_VEL
LIN {X 0,Y 441.263,Z 329.001,A -85,B 0,C 180,E1 -9069.247,E2 -9069.247} C_VEL
LIN {X 0,Y 440.568,Z 342.181,A -85,B 0,C 180,E1 -9071.663,E2 -9071.663} C_VEL
LIN {X 0,Y 444.247,Z 364.829,A -85,B 0,C 180,E1 -9072.229,E2 -9072.229} C_VEL
LIN {X 0,Y 444.231,Z 384.716,A -85,B 0,C 180,E1 -9072.565,E2 -9072.565} C_VEL
LIN {X 0,Y 443.517,Z 450.599,A -85,B 0,C 180,E1 -9073.666,E2 -9073.666} C_VEL
LIN {X 0,Y 443.022,Z 463.857,A -85,B 0,C 180,E1 -9074.061,E2 -9074.061} C_VEL
LIN {X 0,Y 442.469,Z 476.573,A -85,B 0,C 180,E1 -9074.631,E2 -9074.631} C_VEL
LIN {X 0,Y 441.783,Z 488.696,A -85,B 0,C 180,E1 -9075.374,E2 -9075.374} C_VEL
LIN {X 0,Y 441.084,Z 500.531,A -85,B 0,C 180,E1 -9076.319,E2 -9076.319} C_VEL
LIN {X 0,Y 440.474,Z 510.624,A -85,B 0,C 180,E1 -9077.328,E2 -9077.328} C_VEL
LIN {X 0,Y 439.871,Z 520.002,A -85,B 0,C 180,E1 -9078.481,E2 -9078.481} C_VEL
LIN {X 0,Y 439.216,Z 529.072,A -85,B 0,C 180,E1 -9079.864,E2 -9079.864} C_VEL
LIN {X 0,Y 438.844,Z 536.4,A -85,B 0,C 180,E1 -9081.25,E2 -9081.25} C_VEL
LIN {X 0,Y 438.582,Z 542.287,A -85,B 0,C 180,E1 -9082.636,E2 -9082.636} C_VEL
LIN {X 0,Y 438.369,Z 546.865,A -85,B 0,C 180,E1 -9083.997,E2 -9083.997} C_VEL
LIN {X 0,Y 438.341,Z 550.483,A -85,B 0,C 180,E1 -9085.403,E2 -9085.403} C_VEL
LIN {X 0,Y 438.281,Z 552.29,A -85,B 0,C 180,E1 -9086.324,E2 -9086.324} C_VEL
LIN {X 0,Y 438.34,Z 553.661,A -85,B 0,C 180,E1 -9087.244,E2 -9087.244} C_VEL
LIN {X 0,Y 438.295,Z 554.634,A -85,B 0,C 180,E1 -9088.164,E2 -9088.164} C_VEL
LIN {X 0,Y 438.254,Z 555.218,A -85,B 0,C 180,E1 -9089.083,E2 -9089.083} C_VEL
LIN {X 0,Y 438.281,Z 555.384,A -85,B 0,C 180,E1 -9090.001,E2 -9090.001} C_VEL
LIN {X 0,Y 438.296,Z 554.498,A -85,B 0,C 180,E1 -9091.839,E2 -9091.839} C_VEL
LIN {X 0,Y 438.359,Z 553.472,A -85,B 0,C 180,E1 -9092.758,E2 -9092.758} C_VEL
LIN {X 0,Y 438.285,Z 552.007,A -85,B 0,C 180,E1 -9093.679,E2 -9093.679} C_VEL
LIN {X 0,Y 438.384,Z 549.002,A -85,B 0,C 180,E1 -9095.06,E2 -9095.06} C_VEL
LIN {X 0,Y 438.45,Z 544.932,A -85,B 0,C 180,E1 -9096.444,E2 -9096.444} C_VEL
LIN {X 0,Y 438.675,Z 538.668,A -85,B 0,C 180,E1 -9098.06,E2 -9098.06} C_VEL
LIN {X 0,Y 438.975,Z 531.84,A -85,B 0,C 180,E1 -9099.446,E2 -9099.446} C_VEL
LIN {X 0,Y 439.407,Z 523.339,A -85,B 0,C 180,E1 -9100.833,E2 -9100.833} C_VEL
LIN {X 0,Y 439.953,Z 514.579,A -85,B 0,C 180,E1 -9101.987,E2 -9101.987} C_VEL
LIN {X 0,Y 440.549,Z 504.74,A -85,B 0,C 180,E1 -9103.047,E2 -9103.047} C_VEL
LIN {X 0,Y 441.119,Z 493.028,A -85,B 0,C 180,E1 -9104.063,E2 -9104.063} C_VEL
LIN {X 0,Y 441.763,Z 480.959,A -85,B 0,C 180,E1 -9104.866,E2 -9104.866} C_VEL
LIN {X 0,Y 442.311,Z 468.372,A -85,B 0,C 180,E1 -9105.495,E2 -9105.495} C_VEL
LIN {X 0,Y 442.775,Z 456.238,A -85,B 0,C 180,E1 -9105.921,E2 -9105.921} C_VEL
LIN {X 0,Y 443,Z 442.717,A -85,B 0,C 180,E1 -9106.209,E2 -9106.209} C_VEL
LIN {X 0,Y 443.616,Z 364.6,A -85,B 0,C 180,E1 -9107.481,E2 -9107.481} C_VEL
LIN {X 0,Y 440.286,Z 342.531,A -85,B 0,C 180,E1 -9107.981,E2 -9107.981} C_VEL
LIN {X 0,Y 441.205,Z 324.539,A -85,B 0,C 180,E1 -9111.248,E2 -9111.248} C_VEL
LIN {X 0,Y 441.964,Z 309.964,A -85,B 0,C 180,E1 -9113.923,E2 -9113.923} C_VEL
LIN {X 0,Y 440.691,Z 301.873,A -85,B 0,C 180,E1 -9115.506,E2 -9115.506} C_VEL
LIN {X 0,Y 439.465,Z 295.745,A -85,B 0,C 180,E1 -9116.763,E2 -9116.763} C_VEL
LIN {X 0,Y 439.387,Z 295.752,A -85,B 0,C 180,E1 -9119.727,E2 -9119.727} C_VEL
LIN {X 0,Y 439.377,Z 295.75,A -85,B 0,C 180,E1 -9122.947,E2 -9122.947} C_VEL
LIN {X 0,Y 439.379,Z 295.757,A -85,B 0,C 180,E1 -9126.288,E2 -9126.288} C_VEL
LIN {X 0,Y 439.408,Z 295.747,A -85,B 0,C 180,E1 -9129.85,E2 -9129.85} C_VEL
LIN {X 0,Y 439.387,Z 295.755,A -85,B 0,C 180,E1 -9132.627,E2 -9132.627} C_VEL
LIN {X 0,Y 439.406,Z 295.747,A -85,B 0,C 180,E1 -9135.271,E2 -9135.271} C_VEL
LIN {X 0,Y 439.395,Z 295.756,A -85,B 0,C 180,E1 -9138.744,E2 -9138.744} C_VEL
LIN {X 0,Y 439.379,Z 295.749,A -85,B 0,C 180,E1 -9141.608,E2 -9141.608} C_VEL
LIN {X 0,Y 439.402,Z 295.753,A -85,B 0,C 180,E1 -9144.844,E2 -9144.844} C_VEL
LIN {X 0,Y 439.375,Z 295.749,A -85,B 0,C 180,E1 -9148.139,E2 -9148.139} C_VEL
LIN {X 0,Y 439.439,Z 295.744,A -85,B 0,C 180,E1 -9151.598,E2 -9151.598} C_VEL
LIN {X 0,Y 439.406,Z 295.746,A -85,B 0,C 180,E1 -9154.415,E2 -9154.415} C_VEL
LIN {X 0,Y 439.371,Z 295.758,A -85,B 0,C 180,E1 -9157.425,E2 -9157.425} C_VEL
LIN {X 0,Y 439.447,Z 295.741,A -85,B 0,C 180,E1 -9160.663,E2 -9160.663} C_VEL
LIN {X 0,Y 439.468,Z 295.739,A -85,B 0,C 180,E1 -9164.225,E2 -9164.225} C_VEL
LIN {X 0,Y 439.489,Z 295.74,A -85,B 0,C 180,E1 -9168.001,E2 -9168.001} C_VEL
LIN {X 0,Y 439.539,Z 295.736,A -85,B 0,C 180,E1 -9171.726,E2 -9171.726} C_VEL
LIN {X 0,Y 439.614,Z 295.721,A -85,B 0,C 180,E1 -9174.495,E2 -9174.495} C_VEL
LIN {X 0,Y 439.639,Z 295.723,A -85,B 0,C 180,E1 -9178.168,E2 -9178.168} C_VEL
LIN {X 0,Y 439.765,Z 295.708,A -85,B 0,C 180,E1 -9180,E2 -9180} C_VEL
LIN {X 0,Y 439.644,Z 295.718,A -85,B 0,C 180,E1 -9182.749,E2 -9182.749} C_VEL
LIN {X 0,Y 439.609,Z 295.727,A -85,B 0,C 180,E1 -9186.425,E2 -9186.425} C_VEL
LIN {X 0,Y 439.5,Z 295.734,A -85,B 0,C 180,E1 -9189.201,E2 -9189.201} C_VEL
LIN {X 0,Y 439.471,Z 295.74,A -85,B 0,C 180,E1 -9192.937,E2 -9192.937} C_VEL
LIN {X 0,Y 439.452,Z 295.744,A -85,B 0,C 180,E1 -9196.348,E2 -9196.348} C_VEL
LIN {X 0,Y 439.407,Z 295.745,A -85,B 0,C 180,E1 -9199.626,E2 -9199.626} C_VEL
LIN {X 0,Y 439.37,Z 295.755,A -85,B 0,C 180,E1 -9202.575,E2 -9202.575} C_VEL
LIN {X 0,Y 439.41,Z 295.746,A -85,B 0,C 180,E1 -9205.584,E2 -9205.584} C_VEL
LIN {X 0,Y 439.422,Z 295.747,A -85,B 0,C 180,E1 -9208.673,E2 -9208.673} C_VEL
LIN {X 0,Y 439.374,Z 295.75,A -85,B 0,C 180,E1 -9212.03,E2 -9212.03} C_VEL
LIN {X 0,Y 439.397,Z 295.754,A -85,B 0,C 180,E1 -9215.339,E2 -9215.339} C_VEL
LIN {X 0,Y 439.387,Z 295.748,A -85,B 0,C 180,E1 -9218.594,E2 -9218.594} C_VEL
LIN {X 0,Y 439.393,Z 295.753,A -85,B 0,C 180,E1 -9221.256,E2 -9221.256} C_VEL
LIN {X 0,Y 439.403,Z 295.746,A -85,B 0,C 180,E1 -9224.729,E2 -9224.729} C_VEL
LIN {X 0,Y 439.399,Z 295.753,A -85,B 0,C 180,E1 -9227.795,E2 -9227.795} C_VEL
LIN {X 0,Y 439.398,Z 295.749,A -85,B 0,C 180,E1 -9230.223,E2 -9230.223} C_VEL
LIN {X 0,Y 439.377,Z 295.755,A -85,B 0,C 180,E1 -9233.712,E2 -9233.712} C_VEL
LIN {X 0,Y 439.376,Z 295.749,A -85,B 0,C 180,E1 -9237.053,E2 -9237.053} C_VEL
LIN {X 0,Y 439.386,Z 295.754,A -85,B 0,C 180,E1 -9240.273,E2 -9240.273} C_VEL
LIN {X 0,Y 439.431,Z 295.743,A -85,B 0,C 180,E1 -9243.395,E2 -9243.395} C_VEL
LIN {X 0,Y 439.388,Z 295.754,A -85,B 0,C 180,E1 -9246.428,E2 -9246.428} C_VEL
LIN {X 0,Y 439.391,Z 295.747,A -85,B 0,C 180,E1 -9249.396,E2 -9249.396} C_VEL
LIN {X 0,Y 439.433,Z 295.748,A -85,B 0,C 180,E1 -9252.308,E2 -9252.308} C_VEL
LIN {X 0,Y 439.45,Z 295.741,A -85,B 0,C 180,E1 -9255.173,E2 -9255.173} C_VEL
LIN {X 0,Y 439.485,Z 295.737,A -85,B 0,C 180,E1 -9258,E2 -9258} C_VEL
LIN {X 0,Y 439.505,Z 295.737,A -85,B 0,C 180,E1 -9261.724,E2 -9261.724} C_VEL
LIN {X 0,Y 439.631,Z 295.915,A -85,B 0,C 180,E1 -9263.689,E2 -9263.689} C_VEL
LIN {X 0,Y 440.798,Z 303.811,A -85,B 0,C 180,E1 -9265.426,E2 -9265.426} C_VEL
LIN {X 0,Y 440.583,Z 311.86,A -85,B 0,C 180,E1 -9267.113,E2 -9267.113} C_VEL
LIN {X 0,Y 444,Z 330.557,A -85,B 0,C 180,E1 -9267.552,E2 -9267.552} C_VEL
LIN {X 0,Y 443.914,Z 338.275,A -85,B 0,C 180,E1 -9267.678,E2 -9267.678} C_VEL
LIN {X 0,Y 443.271,Z 344.112,A -85,B 0,C 180,E1 -9267.751,E2 -9267.751} C_VEL
LIN {X 0,Y 437.462,Z 363.07,A -85,B 0,C 180,E1 -9267.858,E2 -9267.858} C_VEL
LIN {X 0,Y 436.708,Z 368.913,A -85,B 0,C 180,E1 -9267.93,E2 -9267.93} C_VEL
LIN {X 0,Y 436.136,Z 419.688,A -85,B 0,C 180,E1 -9268.789,E2 -9268.789} C_VEL
LIN {X 0,Y 435.778,Z 432.842,A -85,B 0,C 180,E1 -9269.197,E2 -9269.197} C_VEL
LIN {X 0,Y 435.411,Z 445.219,A -85,B 0,C 180,E1 -9269.767,E2 -9269.767} C_VEL
LIN {X 0,Y 434.94,Z 456.441,A -85,B 0,C 180,E1 -9270.462,E2 -9270.462} C_VEL
LIN {X 0,Y 434.255,Z 468.064,A -85,B 0,C 180,E1 -9271.39,E2 -9271.39} C_VEL
LIN {X 0,Y 433.564,Z 478.522,A -85,B 0,C 180,E1 -9272.437,E2 -9272.437} C_VEL
LIN {X 0,Y 433.101,Z 487.042,A -85,B 0,C 180,E1 -9273.487,E2 -9273.487} C_VEL
LIN {X 0,Y 432.586,Z 494.928,A -85,B 0,C 180,E1 -9274.658,E2 -9274.658} C_VEL
LIN {X 0,Y 432.121,Z 502.635,A -85,B 0,C 180,E1 -9276.067,E2 -9276.067} C_VEL
LIN {X 0,Y 431.845,Z 508.812,A -85,B 0,C 180,E1 -9277.479,E2 -9277.479} C_VEL
LIN {X 0,Y 431.543,Z 513.74,A -85,B 0,C 180,E1 -9278.899,E2 -9278.899} C_VEL
LIN {X 0,Y 431.401,Z 517.531,A -85,B 0,C 180,E1 -9280.322,E2 -9280.322} C_VEL
LIN {X 0,Y 431.229,Z 520.804,A -85,B 0,C 180,E1 -9282.081,E2 -9282.081} C_VEL
LIN {X 0,Y 431.13,Z 522.083,A -85,B 0,C 180,E1 -9283.191,E2 -9283.191} C_VEL
LIN {X 0,Y 431.095,Z 522.747,A -85,B 0,C 180,E1 -9284.153,E2 -9284.153} C_VEL
LIN {X 0,Y 431.153,Z 522.903,A -85,B 0,C 180,E1 -9285.903,E2 -9285.903} C_VEL
LIN {X 0,Y 431.124,Z 522.211,A -85,B 0,C 180,E1 -9287.062,E2 -9287.062} C_VEL
LIN {X 0,Y 431.204,Z 521.184,A -85,B 0,C 180,E1 -9288.038,E2 -9288.038} C_VEL
LIN {X 0,Y 431.341,Z 519.567,A -85,B 0,C 180,E1 -9289.089,E2 -9289.089} C_VEL
LIN {X 0,Y 431.495,Z 516.572,A -85,B 0,C 180,E1 -9290.497,E2 -9290.497} C_VEL
LIN {X 0,Y 431.757,Z 512.262,A -85,B 0,C 180,E1 -9291.985,E2 -9291.985} C_VEL
LIN {X 0,Y 432.112,Z 506.623,A -85,B 0,C 180,E1 -9293.481,E2 -9293.481} C_VEL
LIN {X 0,Y 432.63,Z 499.455,A -85,B 0,C 180,E1 -9294.982,E2 -9294.982} C_VEL
LIN {X 0,Y 433.187,Z 492.033,A -85,B 0,C 180,E1 -9296.236,E2 -9296.236} C_VEL
LIN {X 0,Y 433.831,Z 482.873,A -85,B 0,C 180,E1 -9297.495,E2 -9297.495} C_VEL
LIN {X 0,Y 434.527,Z 472.668,A -85,B 0,C 180,E1 -9298.628,E2 -9298.628} C_VEL
LIN {X 0,Y 435.321,Z 461.186,A -85,B 0,C 180,E1 -9299.644,E2 -9299.644} C_VEL
LIN {X 0,Y 435.94,Z 449.437,A -85,B 0,C 180,E1 -9300.45,E2 -9300.45} C_VEL
LIN {X 0,Y 436.476,Z 437.237,A -85,B 0,C 180,E1 -9301.083,E2 -9301.083} C_VEL
LIN {X 0,Y 436.86,Z 424.057,A -85,B 0,C 180,E1 -9301.561,E2 -9301.561} C_VEL
LIN {X 0,Y 437.213,Z 408.101,A -85,B 0,C 180,E1 -9301.884,E2 -9301.884} C_VEL
LIN {X 0,Y 438.027,Z 330.407,A -85,B 0,C 180,E1 -9303.186,E2 -9303.186} C_VEL
LIN {X 0,Y 434.371,Z 313.635,A -85,B 0,C 180,E1 -9303.664,E2 -9303.664} C_VEL
LIN {X 0,Y 434.03,Z 312.03,A -85,B 0,C 180,E1 -9303.729,E2 -9303.729} C_VEL
LIN {X 0,Y 434.112,Z 305.563,A -85,B 0,C 180,E1 -9305.078,E2 -9305.078} C_VEL
LIN {X 0,Y 432.28,Z 296.641,A -85,B 0,C 180,E1 -9307.11,E2 -9307.11} C_VEL
LIN {X 0,Y 432.277,Z 296.639,A -85,B 0,C 180,E1 -9310.171,E2 -9310.171} C_VEL
LIN {X 0,Y 432.289,Z 296.639,A -85,B 0,C 180,E1 -9313.062,E2 -9313.062} C_VEL
LIN {X 0,Y 432.321,Z 296.629,A -85,B 0,C 180,E1 -9315.664,E2 -9315.664} C_VEL
LIN {X 0,Y 432.298,Z 296.634,A -85,B 0,C 180,E1 -9318.4,E2 -9318.4} C_VEL
LIN {X 0,Y 432.309,Z 296.638,A -85,B 0,C 180,E1 -9321.847,E2 -9321.847} C_VEL
LIN {X 0,Y 432.322,Z 296.622,A -85,B 0,C 180,E1 -9325.322,E2 -9325.322} C_VEL
LIN {X 0,Y 432.306,Z 296.629,A -85,B 0,C 180,E1 -9328.653,E2 -9328.653} C_VEL
LIN {X 0,Y 432.333,Z 296.631,A -85,B 0,C 180,E1 -9331.873,E2 -9331.873} C_VEL
LIN {X 0,Y 432.363,Z 296.624,A -85,B 0,C 180,E1 -9335.538,E2 -9335.538} C_VEL
LIN {X 0,Y 432.335,Z 296.623,A -85,B 0,C 180,E1 -9339.045,E2 -9339.045} C_VEL
LIN {X 0,Y 432.358,Z 296.63,A -85,B 0,C 180,E1 -9342.01,E2 -9342.01} C_VEL
LIN {X 0,Y 432.378,Z 296.622,A -85,B 0,C 180,E1 -9344.926,E2 -9344.926} C_VEL
LIN {X 0,Y 432.444,Z 296.614,A -85,B 0,C 180,E1 -9347.803,E2 -9347.803} C_VEL
LIN {X 0,Y 432.468,Z 296.611,A -85,B 0,C 180,E1 -9351.59,E2 -9351.59} C_VEL
LIN {X 0,Y 432.569,Z 296.601,A -85,B 0,C 180,E1 -9354.406,E2 -9354.406} C_VEL
LIN {X 0,Y 432.59,Z 296.594,A -85,B 0,C 180,E1 -9358.138,E2 -9358.138} C_VEL
LIN {X 0,Y 432.717,Z 296.579,A -85,B 0,C 180,E1 -9360,E2 -9360} C_VEL
LIN {X 0,Y 432.578,Z 296.593,A -85,B 0,C 180,E1 -9362.794,E2 -9362.794} C_VEL
LIN {X 0,Y 432.554,Z 296.606,A -85,B 0,C 180,E1 -9366.531,E2 -9366.531} C_VEL
LIN {X 0,Y 432.43,Z 296.614,A -85,B 0,C 180,E1 -9369.354,E2 -9369.354} C_VEL
LIN {X 0,Y 432.417,Z 296.617,A -85,B 0,C 180,E1 -9372.804,E2 -9372.804} C_VEL
LIN {X 0,Y 432.399,Z 296.622,A -85,B 0,C 180,E1 -9376.48,E2 -9376.48} C_VEL
LIN {X 0,Y 432.325,Z 296.627,A -85,B 0,C 180,E1 -9379.961,E2 -9379.961} C_VEL
LIN {X 0,Y 432.306,Z 296.632,A -85,B 0,C 180,E1 -9382.965,E2 -9382.965} C_VEL
LIN {X 0,Y 432.353,Z 296.626,A -85,B 0,C 180,E1 -9386.033,E2 -9386.033} C_VEL
LIN {X 0,Y 432.341,Z 296.63,A -85,B 0,C 180,E1 -9389.188,E2 -9389.188} C_VEL
LIN {X 0,Y 432.322,Z 296.625,A -85,B 0,C 180,E1 -9392.296,E2 -9392.296} C_VEL
LIN {X 0,Y 432.331,Z 296.631,A -85,B 0,C 180,E1 -9394.678,E2 -9394.678} C_VEL
LIN {X 0,Y 432.343,Z 296.629,A -85,B 0,C 180,E1 -9398.15,E2 -9398.15} C_VEL
LIN {X 0,Y 432.358,Z 296.629,A -85,B 0,C 180,E1 -9401.609,E2 -9401.609} C_VEL
LIN {X 0,Y 432.333,Z 296.628,A -85,B 0,C 180,E1 -9404.348,E2 -9404.348} C_VEL
LIN {X 0,Y 432.358,Z 296.622,A -85,B 0,C 180,E1 -9407.011,E2 -9407.011} C_VEL
LIN {X 0,Y 432.35,Z 296.625,A -85,B 0,C 180,E1 -9409.819,E2 -9409.819} C_VEL
LIN {X 0,Y 432.311,Z 296.633,A -85,B 0,C 180,E1 -9413.025,E2 -9413.025} C_VEL
LIN {X 0,Y 432.354,Z 296.628,A -85,B 0,C 180,E1 -9415.998,E2 -9415.998} C_VEL
LIN {X 0,Y 432.343,Z 296.631,A -85,B 0,C 180,E1 -9419.491,E2 -9419.491} C_VEL
LIN {X 0,Y 432.439,Z 296.741,A -85,B 0,C 180,E1 -9422.475,E2 -9422.475} C_VEL
LIN {X 0,Y 434.781,Z 307.896,A -85,B 0,C 180,E1 -9424.852,E2 -9424.852} C_VEL
LIN {X 0,Y 435.422,Z 313.325,A -85,B 0,C 180,E1 -9425.951,E2 -9425.951} C_VEL
LIN {X 0,Y 434.332,Z 330.25,A -85,B 0,C 180,E1 -9429.148,E2 -9429.148} C_VEL
LIN {X 0,Y 433.69,Z 341.848,A -85,B 0,C 180,E1 -9431.311,E2 -9431.311} C_VEL
LIN {X 0,Y 437.388,Z 363.996,A -85,B 0,C 180,E1 -9431.891,E2 -9431.891} C_VEL
LIN {X 0,Y 437.719,Z 370.068,A -85,B 0,C 180,E1 -9432.012,E2 -9432.012} C_VEL
LIN {X 0,Y 436.793,Z 450.563,A -85,B 0,C 180,E1 -9433.377,E2 -9433.377} C_VEL
LIN {X 0,Y 436.269,Z 463.727,A -85,B 0,C 180,E1 -9433.777,E2 -9433.777} C_VEL
LIN {X 0,Y 435.652,Z 476.946,A -85,B 0,C 180,E1 -9434.385,E2 -9434.385} C_VEL
LIN {X 0,Y 434.913,Z 488.866,A -85,B 0,C 180,E1 -9435.137,E2 -9435.137} C_VEL
LIN {X 0,Y 434.157,Z 501.007,A -85,B 0,C 180,E1 -9436.134,E2 -9436.134} C_VEL
LIN {X 0,Y 433.531,Z 510.627,A -85,B 0,C 180,E1 -9437.122,E2 -9437.122} C_VEL
LIN {X 0,Y 432.908,Z 519.94,A -85,B 0,C 180,E1 -9438.293,E2 -9438.293} C_VEL
LIN {X 0,Y 432.186,Z 528.976,A -85,B 0,C 180,E1 -9439.697,E2 -9439.697} C_VEL
LIN {X 0,Y 431.808,Z 536.274,A -85,B 0,C 180,E1 -9441.107,E2 -9441.107} C_VEL
LIN {X 0,Y 431.517,Z 542.134,A -85,B 0,C 180,E1 -9442.515,E2 -9442.515} C_VEL
LIN {X 0,Y 431.326,Z 546.04,A -85,B 0,C 180,E1 -9443.687,E2 -9443.687} C_VEL
LIN {X 0,Y 431.27,Z 550.285,A -85,B 0,C 180,E1 -9445.328,E2 -9445.328} C_VEL
LIN {X 0,Y 431.188,Z 552.07,A -85,B 0,C 180,E1 -9446.263,E2 -9446.263} C_VEL
LIN {X 0,Y 431.236,Z 553.43,A -85,B 0,C 180,E1 -9447.199,E2 -9447.199} C_VEL
LIN {X 0,Y 431.218,Z 554.393,A -85,B 0,C 180,E1 -9448.133,E2 -9448.133} C_VEL
LIN {X 0,Y 431.171,Z 554.967,A -85,B 0,C 180,E1 -9449.067,E2 -9449.067} C_VEL
LIN {X 0,Y 431.193,Z 555.114,A -85,B 0,C 180,E1 -9450.001,E2 -9450.001} C_VEL
LIN {X 0,Y 431.219,Z 554.209,A -85,B 0,C 180,E1 -9451.869,E2 -9451.869} C_VEL
LIN {X 0,Y 431.268,Z 553.173,A -85,B 0,C 180,E1 -9452.804,E2 -9452.804} C_VEL
LIN {X 0,Y 431.192,Z 551.687,A -85,B 0,C 180,E1 -9453.739,E2 -9453.739} C_VEL
LIN {X 0,Y 431.294,Z 548.66,A -85,B 0,C 180,E1 -9455.143,E2 -9455.143} C_VEL
LIN {X 0,Y 431.378,Z 544.563,A -85,B 0,C 180,E1 -9456.55,E2 -9456.55} C_VEL
LIN {X 0,Y 431.605,Z 538.268,A -85,B 0,C 180,E1 -9458.193,E2 -9458.193} C_VEL
LIN {X 0,Y 431.921,Z 531.408,A -85,B 0,C 180,E1 -9459.602,E2 -9459.602} C_VEL
LIN {X 0,Y 432.408,Z 522.856,A -85,B 0,C 180,E1 -9461.011,E2 -9461.011} C_VEL
LIN {X 0,Y 432.966,Z 514.05,A -85,B 0,C 180,E1 -9462.183,E2 -9462.183} C_VEL
LIN {X 0,Y 433.6,Z 503.738,A -85,B 0,C 180,E1 -9463.302,E2 -9463.302} C_VEL
LIN {X 0,Y 434.17,Z 492.345,A -85,B 0,C 180,E1 -9464.293,E2 -9464.293} C_VEL
LIN {X 0,Y 434.844,Z 480.152,A -85,B 0,C 180,E1 -9465.108,E2 -9465.108} C_VEL
LIN {X 0,Y 435.403,Z 467.398,A -85,B 0,C 180,E1 -9465.747,E2 -9465.747} C_VEL
LIN {X 0,Y 435.918,Z 454.799,A -85,B 0,C 180,E1 -9466.179,E2 -9466.179} C_VEL
LIN {X 0,Y 436.246,Z 438.762,A -85,B 0,C 180,E1 -9466.497,E2 -9466.497} C_VEL
LIN {X 0,Y 436.794,Z 365.414,A -85,B 0,C 180,E1 -9467.712,E2 -9467.712} C_VEL
LIN {X 0,Y 433.353,Z 342.326,A -85,B 0,C 180,E1 -9468.232,E2 -9468.232} C_VEL
LIN {X 0,Y 434.284,Z 324.067,A -85,B 0,C 180,E1 -9471.604,E2 -9471.604} C_VEL
LIN {X 0,Y 435.001,Z 310.813,A -85,B 0,C 180,E1 -9474.077,E2 -9474.077} C_VEL
LIN {X 0,Y 433.366,Z 301.337,A -85,B 0,C 180,E1 -9475.969,E2 -9475.969} C_VEL
LIN {X 0,Y 432.455,Z 296.617,A -85,B 0,C 180,E1 -9476.944,E2 -9476.944} C_VEL
LIN {X 0,Y 432.353,Z 296.632,A -85,B 0,C 180,E1 -9480.511,E2 -9480.511} C_VEL
LIN {X 0,Y 432.364,Z 296.628,A -85,B 0,C 180,E1 -9484.004,E2 -9484.004} C_VEL
LIN {X 0,Y 432.327,Z 296.628,A -85,B 0,C 180,E1 -9487.197,E2 -9487.197} C_VEL
LIN {X 0,Y 432.331,Z 296.634,A -85,B 0,C 180,E1 -9490.561,E2 -9490.561} C_VEL
LIN {X 0,Y 432.322,Z 296.63,A -85,B 0,C 180,E1 -9493.062,E2 -9493.062} C_VEL
LIN {X 0,Y 432.339,Z 296.626,A -85,B 0,C 180,E1 -9495.665,E2 -9495.665} C_VEL
LIN {X 0,Y 432.339,Z 296.63,A -85,B 0,C 180,E1 -9498.398,E2 -9498.398} C_VEL
LIN {X 0,Y 432.342,Z 296.625,A -85,B 0,C 180,E1 -9501.85,E2 -9501.85} C_VEL
LIN {X 0,Y 432.334,Z 296.63,A -85,B 0,C 180,E1 -9505.322,E2 -9505.322} C_VEL
LIN {X 0,Y 432.325,Z 296.631,A -85,B 0,C 180,E1 -9508.654,E2 -9508.654} C_VEL
LIN {X 0,Y 432.388,Z 296.621,A -85,B 0,C 180,E1 -9511.877,E2 -9511.877} C_VEL
LIN {X 0,Y 432.354,Z 296.628,A -85,B 0,C 180,E1 -9514.999,E2 -9514.999} C_VEL
LIN {X 0,Y 432.364,Z 296.624,A -85,B 0,C 180,E1 -9518.046,E2 -9518.046} C_VEL
LIN {X 0,Y 432.39,Z 296.622,A -85,B 0,C 180,E1 -9521.03,E2 -9521.03} C_VEL
LIN {X 0,Y 432.436,Z 296.617,A -85,B 0,C 180,E1 -9523.961,E2 -9523.961} C_VEL
LIN {X 0,Y 432.465,Z 296.617,A -85,B 0,C 180,E1 -9527.803,E2 -9527.803} C_VEL
LIN {X 0,Y 432.488,Z 296.612,A -85,B 0,C 180,E1 -9531.59,E2 -9531.59} C_VEL
LIN {X 0,Y 432.587,Z 296.597,A -85,B 0,C 180,E1 -9534.406,E2 -9534.406} C_VEL
LIN {X 0,Y 432.609,Z 296.599,A -85,B 0,C 180,E1 -9538.138,E2 -9538.138} C_VEL
LIN {X 0,Y 432.735,Z 296.584,A -85,B 0,C 180,E1 -9540,E2 -9540} C_VEL
LIN {X 0,Y 432.595,Z 296.595,A -85,B 0,C 180,E1 -9542.793,E2 -9542.793} C_VEL
LIN {X 0,Y 432.596,Z 296.595,A -85,B 0,C 180,E1 -9545.594,E2 -9545.594} C_VEL
LIN {X 0,Y 432.469,Z 296.618,A -85,B 0,C 180,E1 -9548.41,E2 -9548.41} C_VEL
LIN {X 0,Y 432.464,Z 296.614,A -85,B 0,C 180,E1 -9552.196,E2 -9552.196} C_VEL
LIN {X 0,Y 432.436,Z 296.615,A -85,B 0,C 180,E1 -9556.038,E2 -9556.038} C_VEL
LIN {X 0,Y 432.392,Z 296.62,A -85,B 0,C 180,E1 -9559.484,E2 -9559.484} C_VEL
LIN {X 0,Y 432.324,Z 296.635,A -85,B 0,C 180,E1 -9562.964,E2 -9562.964} C_VEL
LIN {X 0,Y 432.369,Z 296.622,A -85,B 0,C 180,E1 -9566.032,E2 -9566.032} C_VEL
LIN {X 0,Y 432.348,Z 296.632,A -85,B 0,C 180,E1 -9569.187,E2 -9569.187} C_VEL
LIN {X 0,Y 432.327,Z 296.628,A -85,B 0,C 180,E1 -9572.442,E2 -9572.442} C_VEL
LIN {X 0,Y 432.347,Z 296.628,A -85,B 0,C 180,E1 -9575.631,E2 -9575.631} C_VEL
LIN {X 0,Y 432.354,Z 296.632,A -85,B 0,C 180,E1 -9579.342,E2 -9579.342} C_VEL
LIN {X 0,Y 432.338,Z 296.63,A -85,B 0,C 180,E1 -9581.796,E2 -9581.796} C_VEL
LIN {X 0,Y 432.338,Z 296.626,A -85,B 0,C 180,E1 -9584.347,E2 -9584.347} C_VEL
LIN {X 0,Y 432.323,Z 296.629,A -85,B 0,C 180,E1 -9587.015,E2 -9587.015} C_VEL
LIN {X 0,Y 432.338,Z 296.633,A -85,B 0,C 180,E1 -9589.82,E2 -9589.82} C_VEL
LIN {X 0,Y 432.31,Z 296.63,A -85,B 0,C 180,E1 -9593.021,E2 -9593.021} C_VEL
LIN {X 0,Y 432.363,Z 296.631,A -85,B 0,C 180,E1 -9595.996,E2 -9595.996} C_VEL
LIN {X 0,Y 432.351,Z 296.626,A -85,B 0,C 180,E1 -9599.489,E2 -9599.489} C_VEL
LIN {X 0,Y 432.394,Z 296.62,A -85,B 0,C 180,E1 -9602.927,E2 -9602.927} C_VEL
LIN {X 0,Y 432.371,Z 296.627,A -85,B 0,C 180,E1 -9606.022,E2 -9606.022} C_VEL
LIN {X 0,Y 432.353,Z 296.625,A -85,B 0,C 180,E1 -9609.045,E2 -9609.045} C_VEL
LIN {X 0,Y 432.38,Z 296.623,A -85,B 0,C 180,E1 -9612.01,E2 -9612.01} C_VEL
LIN {X 0,Y 432.398,Z 296.622,A -85,B 0,C 180,E1 -9614.925,E2 -9614.925} C_VEL
LIN {X 0,Y 432.461,Z 296.611,A -85,B 0,C 180,E1 -9617.802,E2 -9617.802} C_VEL
LIN {X 0,Y 432.465,Z 296.615,A -85,B 0,C 180,E1 -9621.589,E2 -9621.589} C_VEL
LIN {X 0,Y 432.578,Z 296.712,A -85,B 0,C 180,E1 -9623.498,E2 -9623.498} C_VEL
LIN {X 0,Y 433.824,Z 305.022,A -85,B 0,C 180,E1 -9625.353,E2 -9625.353} C_VEL
LIN {X 0,Y 433.637,Z 312.056,A -85,B 0,C 180,E1 -9626.843,E2 -9626.843} C_VEL
LIN {X 0,Y 437.18,Z 331.4,A -85,B 0,C 180,E1 -9627.315,E2 -9627.315} C_VEL
LIN {X 0,Y 436.708,Z 368.913,A -85,B 0,C 180,E1 -9627.93,E2 -9627.93} C_VEL
LIN {X 0,Y 435.984,Z 374.75,A -85,B 0,C 180,E1 -9628.003,E2 -9628.003} C_VEL
LIN {X 0,Y 430.291,Z 393.72,A -85,B 0,C 180,E1 -9628.124,E2 -9628.124} C_VEL
LIN {X 0,Y 429.551,Z 399.557,A -85,B 0,C 180,E1 -9628.197,E2 -9628.197} C_VEL
LIN {X 0,Y 429.22,Z 421.411,A -85,B 0,C 180,E1 -9628.599,E2 -9628.599} C_VEL
LIN {X 0,Y 428.841,Z 434.71,A -85,B 0,C 180,E1 -9629.038,E2 -9629.038} C_VEL
LIN {X 0,Y 428.416,Z 447.595,A -85,B 0,C 180,E1 -9629.676,E2 -9629.676} C_VEL
LIN {X 0,Y 427.859,Z 459.512,A -85,B 0,C 180,E1 -9630.469,E2 -9630.469} C_VEL
LIN {X 0,Y 427.196,Z 470.615,A -85,B 0,C 180,E1 -9631.413,E2 -9631.413} C_VEL
LIN {X 0,Y 426.572,Z 479.619,A -85,B 0,C 180,E1 -9632.359,E2 -9632.359} C_VEL
LIN {X 0,Y 425.978,Z 488.842,A -85,B 0,C 180,E1 -9633.546,E2 -9633.546} C_VEL
LIN {X 0,Y 425.411,Z 497.803,A -85,B 0,C 180,E1 -9634.974,E2 -9634.974} C_VEL
LIN {X 0,Y 425.038,Z 505.021,A -85,B 0,C 180,E1 -9636.407,E2 -9636.407} C_VEL
LIN {X 0,Y 424.742,Z 509.906,A -85,B 0,C 180,E1 -9637.605,E2 -9637.605} C_VEL
LIN {X 0,Y 424.442,Z 514.663,A -85,B 0,C 180,E1 -9639.049,E2 -9639.049} C_VEL
LIN {X 0,Y 424.306,Z 518.29,A -85,B 0,C 180,E1 -9640.496,E2 -9640.496} C_VEL
LIN {X 0,Y 424.131,Z 521.178,A -85,B 0,C 180,E1 -9642.137,E2 -9642.137} C_VEL
LIN {X 0,Y 424.044,Z 522.537,A -85,B 0,C 180,E1 -9643.415,E2 -9643.415} C_VEL
LIN {X 0,Y 424,Z 523.127,A -85,B 0,C 180,E1 -9644.395,E2 -9644.395} C_VEL
LIN {X 0,Y 424.058,Z 523.152,A -85,B 0,C 180,E1 -9646.004,E2 -9646.004} C_VEL
LIN {X 0,Y 424.052,Z 522.289,A -85,B 0,C 180,E1 -9647.355,E2 -9647.355} C_VEL
LIN {X 0,Y 424.159,Z 521.158,A -85,B 0,C 180,E1 -9648.348,E2 -9648.348} C_VEL
LIN {X 0,Y 424.325,Z 518.59,A -85,B 0,C 180,E1 -9649.847,E2 -9649.847} C_VEL
LIN {X 0,Y 424.544,Z 514.905,A -85,B 0,C 180,E1 -9651.356,E2 -9651.356} C_VEL
LIN {X 0,Y 424.896,Z 509.976,A -85,B 0,C 180,E1 -9652.872,E2 -9652.872} C_VEL
LIN {X 0,Y 425.395,Z 503.636,A -85,B 0,C 180,E1 -9654.393,E2 -9654.393} C_VEL
LIN {X 0,Y 425.993,Z 495.61,A -85,B 0,C 180,E1 -9655.923,E2 -9655.923} C_VEL
LIN {X 0,Y 426.694,Z 486.769,A -85,B 0,C 180,E1 -9657.26,E2 -9657.26} C_VEL
LIN {X 0,Y 427.446,Z 476.847,A -85,B 0,C 180,E1 -9658.476,E2 -9658.476} C_VEL
LIN {X 0,Y 428.203,Z 465.832,A -85,B 0,C 180,E1 -9659.556,E2 -9659.556} C_VEL
LIN {X 0,Y 428.896,Z 455.047,A -85,B 0,C 180,E1 -9660.391,E2 -9660.391} C_VEL
LIN {X 0,Y 429.483,Z 443.389,A -85,B 0,C 180,E1 -9661.095,E2 -9661.095} C_VEL
LIN {X 0,Y 430.022,Z 430.475,A -85,B 0,C 180,E1 -9661.664,E2 -9661.664} C_VEL
LIN {X 0,Y 430.32,Z 418.315,A -85,B 0,C 180,E1 -9662.014,E2 -9662.014} C_VEL
LIN {X 0,Y 431.355,Z 331.082,A -85,B 0,C 180,E1 -9663.511,E2 -9663.511} C_VEL
LIN {X 0,Y 427.579,Z 314.078,A -85,B 0,C 180,E1 -9664.013,E2 -9664.013} C_VEL
LIN {X 0,Y 427.17,Z 312.226,A -85,B 0,C 180,E1 -9664.101,E2 -9664.101} C_VEL
LIN {X 0,Y 427.25,Z 307.283,A -85,B 0,C 180,E1 -9665.148,E2 -9665.148} C_VEL
LIN {X 0,Y 425.268,Z 297.515,A -85,B 0,C 180,E1 -9667.425,E2 -9667.425} C_VEL
LIN {X 0,Y 425.232,Z 297.517,A -85,B 0,C 180,E1 -9670.513,E2 -9670.513} C_VEL
LIN {X 0,Y 425.234,Z 297.52,A -85,B 0,C 180,E1 -9673.348,E2 -9673.348} C_VEL
LIN {X 0,Y 425.246,Z 297.507,A -85,B 0,C 180,E1 -9676.042,E2 -9676.042} C_VEL
LIN {X 0,Y 425.238,Z 297.513,A -85,B 0,C 180,E1 -9678.617,E2 -9678.617} C_VEL
LIN {X 0,Y 425.263,Z 297.512,A -85,B 0,C 180,E1 -9681.098,E2 -9681.098} C_VEL
LIN {X 0,Y 425.283,Z 297.495,A -85,B 0,C 180,E1 -9684.663,E2 -9684.663} C_VEL
LIN {X 0,Y 425.25,Z 297.511,A -85,B 0,C 180,E1 -9688.072,E2 -9688.072} C_VEL
LIN {X 0,Y 425.3,Z 297.507,A -85,B 0,C 180,E1 -9691.366,E2 -9691.366} C_VEL
LIN {X 0,Y 425.256,Z 297.508,A -85,B 0,C 180,E1 -9694.552,E2 -9694.552} C_VEL
LIN {X 0,Y 425.269,Z 297.509,A -85,B 0,C 180,E1 -9696.633,E2 -9696.633} C_VEL
LIN {X 0,Y 425.28,Z 297.505,A -85,B 0,C 180,E1 -9699.694,E2 -9699.694} C_VEL
LIN {X 0,Y 425.324,Z 297.497,A -85,B 0,C 180,E1 -9702.697,E2 -9702.697} C_VEL
LIN {X 0,Y 425.331,Z 297.502,A -85,B 0,C 180,E1 -9705.65,E2 -9705.65} C_VEL
LIN {X 0,Y 425.336,Z 297.5,A -85,B 0,C 180,E1 -9708.564,E2 -9708.564} C_VEL
LIN {X 0,Y 425.422,Z 297.489,A -85,B 0,C 180,E1 -9711.45,E2 -9711.45} C_VEL
LIN {X 0,Y 425.524,Z 297.477,A -85,B 0,C 180,E1 -9714.313,E2 -9714.313} C_VEL
LIN {X 0,Y 425.559,Z 297.469,A -85,B 0,C 180,E1 -9718.107,E2 -9718.107} C_VEL
LIN {X 0,Y 425.687,Z 297.455,A -85,B 0,C 180,E1 -9720,E2 -9720} C_VEL
LIN {X 0,Y 425.531,Z 297.47,A -85,B 0,C 180,E1 -9722.84,E2 -9722.84} C_VEL
LIN {X 0,Y 425.513,Z 297.482,A -85,B 0,C 180,E1 -9726.639,E2 -9726.639} C_VEL
LIN {X 0,Y 425.388,Z 297.49,A -85,B 0,C 180,E1 -9729.51,E2 -9729.51} C_VEL
LIN {X 0,Y 425.379,Z 297.492,A -85,B 0,C 180,E1 -9732.904,E2 -9732.904} C_VEL
LIN {X 0,Y 425.348,Z 297.502,A -85,B 0,C 180,E1 -9736.606,E2 -9736.606} C_VEL
LIN {X 0,Y 425.315,Z 297.501,A -85,B 0,C 180,E1 -9739.637,E2 -9739.637} C_VEL
LIN {X 0,Y 425.294,Z 297.502,A -85,B 0,C 180,E1 -9743.366,E2 -9743.366} C_VEL
LIN {X 0,Y 425.337,Z 297.504,A -85,B 0,C 180,E1 -9746.846,E2 -9746.846} C_VEL
LIN {X 0,Y 425.308,Z 297.506,A -85,B 0,C 180,E1 -9749.719,E2 -9749.719} C_VEL
LIN {X 0,Y 425.274,Z 297.508,A -85,B 0,C 180,E1 -9753.049,E2 -9753.049} C_VEL
LIN {X 0,Y 425.275,Z 297.508,A -85,B 0,C 180,E1 -9755.931,E2 -9755.931} C_VEL
LIN {X 0,Y 425.304,Z 297.508,A -85,B 0,C 180,E1 -9759.047,E2 -9759.047} C_VEL
LIN {X 0,Y 425.307,Z 297.505,A -85,B 0,C 180,E1 -9761.964,E2 -9761.964} C_VEL
LIN {X 0,Y 425.307,Z 297.501,A -85,B 0,C 180,E1 -9765.28,E2 -9765.28} C_VEL
LIN {X 0,Y 425.303,Z 297.505,A -85,B 0,C 180,E1 -9768.627,E2 -9768.627} C_VEL
LIN {X 0,Y 425.315,Z 297.502,A -85,B 0,C 180,E1 -9771.106,E2 -9771.106} C_VEL
LIN {X 0,Y 425.295,Z 297.509,A -85,B 0,C 180,E1 -9774.666,E2 -9774.666} C_VEL
LIN {X 0,Y 425.26,Z 297.512,A -85,B 0,C 180,E1 -9778.075,E2 -9778.075} C_VEL
LIN {X 0,Y 425.328,Z 297.507,A -85,B 0,C 180,E1 -9781.37,E2 -9781.37} C_VEL
LIN {X 0,Y 425.372,Z 297.553,A -85,B 0,C 180,E1 -9782.145,E2 -9782.145} C_VEL
LIN {X 0,Y 427.869,Z 309.397,A -85,B 0,C 180,E1 -9784.72,E2 -9784.72} C_VEL
LIN {X 0,Y 428.543,Z 314.597,A -85,B 0,C 180,E1 -9785.797,E2 -9785.797} C_VEL
LIN {X 0,Y 427.409,Z 331.518,A -85,B 0,C 180,E1 -9789.047,E2 -9789.047} C_VEL
LIN {X 0,Y 426.813,Z 341.623,A -85,B 0,C 180,E1 -9790.965,E2 -9790.965} C_VEL
LIN {X 0,Y 430.707,Z 365.018,A -85,B 0,C 180,E1 -9791.583,E2 -9791.583} C_VEL
LIN {X 0,Y 431.062,Z 369.843,A -85,B 0,C 180,E1 -9791.685,E2 -9791.685} C_VEL
LIN {X 0,Y 430.071,Z 450.601,A -85,B 0,C 180,E1 -9793.079,E2 -9793.079} C_VEL
LIN {X 0,Y 429.48,Z 464.42,A -85,B 0,C 180,E1 -9793.514,E2 -9793.514} C_VEL
LIN {X 0,Y 428.84,Z 477.339,A -85,B 0,C 180,E1 -9794.13,E2 -9794.13} C_VEL
LIN {X 0,Y 428.053,Z 489.097,A -85,B 0,C 180,E1 -9794.893,E2 -9794.893} C_VEL
LIN {X 0,Y 427.327,Z 500.271,A -85,B 0,C 180,E1 -9795.825,E2 -9795.825} C_VEL
LIN {X 0,Y 426.646,Z 509.627,A -85,B 0,C 180,E1 -9796.789,E2 -9796.789} C_VEL
LIN {X 0,Y 426.071,Z 518.209,A -85,B 0,C 180,E1 -9797.861,E2 -9797.861} C_VEL
LIN {X 0,Y 425.393,Z 526.138,A -85,B 0,C 180,E1 -9799.049,E2 -9799.049} C_VEL
LIN {X 0,Y 424.867,Z 533.916,A -85,B 0,C 180,E1 -9800.48,E2 -9800.48} C_VEL
LIN {X 0,Y 424.522,Z 540.163,A -85,B 0,C 180,E1 -9801.912,E2 -9801.912} C_VEL
LIN {X 0,Y 424.3,Z 545.147,A -85,B 0,C 180,E1 -9803.343,E2 -9803.343} C_VEL
LIN {X 0,Y 424.205,Z 549.01,A -85,B 0,C 180,E1 -9804.773,E2 -9804.773} C_VEL
LIN {X 0,Y 424.099,Z 551.851,A -85,B 0,C 180,E1 -9806.201,E2 -9806.201} C_VEL
LIN {X 0,Y 424.133,Z 553.2,A -85,B 0,C 180,E1 -9807.152,E2 -9807.152} C_VEL
LIN {X 0,Y 424.143,Z 554.155,A -85,B 0,C 180,E1 -9808.102,E2 -9808.102} C_VEL
LIN {X 0,Y 424.091,Z 554.715,A -85,B 0,C 180,E1 -9809.052,E2 -9809.052} C_VEL
LIN {X 0,Y 424.109,Z 554.844,A -85,B 0,C 180,E1 -9810.001,E2 -9810.001} C_VEL
LIN {X 0,Y 424.145,Z 553.919,A -85,B 0,C 180,E1 -9811.9,E2 -9811.9} C_VEL
LIN {X 0,Y 424.164,Z 552.87,A -85,B 0,C 180,E1 -9812.851,E2 -9812.851} C_VEL
LIN {X 0,Y 424.103,Z 551.363,A -85,B 0,C 180,E1 -9813.802,E2 -9813.802} C_VEL
LIN {X 0,Y 424.207,Z 548.312,A -85,B 0,C 180,E1 -9815.229,E2 -9815.229} C_VEL
LIN {X 0,Y 424.301,Z 544.19,A -85,B 0,C 180,E1 -9816.66,E2 -9816.66} C_VEL
LIN {X 0,Y 424.537,Z 537.868,A -85,B 0,C 180,E1 -9818.33,E2 -9818.33} C_VEL
LIN {X 0,Y 424.89,Z 530.978,A -85,B 0,C 180,E1 -9819.763,E2 -9819.763} C_VEL
LIN {X 0,Y 425.277,Z 523.941,A -85,B 0,C 180,E1 -9820.957,E2 -9820.957} C_VEL
LIN {X 0,Y 425.88,Z 515.465,A -85,B 0,C 180,E1 -9822.147,E2 -9822.147} C_VEL
LIN {X 0,Y 426.555,Z 504.975,A -85,B 0,C 180,E1 -9823.338,E2 -9823.338} C_VEL
LIN {X 0,Y 427.155,Z 493.136,A -85,B 0,C 180,E1 -9824.411,E2 -9824.411} C_VEL
LIN {X 0,Y 427.868,Z 481.288,A -85,B 0,C 180,E1 -9825.238,E2 -9825.238} C_VEL
LIN {X 0,Y 428.472,Z 468.952,A -85,B 0,C 180,E1 -9825.887,E2 -9825.887} C_VEL
LIN {X 0,Y 428.995,Z 456.348,A -85,B 0,C 180,E1 -9826.355,E2 -9826.355} C_VEL
LIN {X 0,Y 429.254,Z 443.385,A -85,B 0,C 180,E1 -9826.651,E2 -9826.651} C_VEL
LIN {X 0,Y 429.927,Z 366.17,A -85,B 0,C 180,E1 -9827.947,E2 -9827.947} C_VEL
LIN {X 0,Y 426.365,Z 342.058,A -85,B 0,C 180,E1 -9828.501,E2 -9828.501} C_VEL
LIN {X 0,Y 427.368,Z 323.576,A -85,B 0,C 180,E1 -9831.971,E2 -9831.971} C_VEL
LIN {X 0,Y 427.997,Z 311.626,A -85,B 0,C 180,E1 -9834.239,E2 -9834.239} C_VEL
LIN {X 0,Y 426.314,Z 302.135,A -85,B 0,C 180,E1 -9836.168,E2 -9836.168} C_VEL
LIN {X 0,Y 425.407,Z 297.495,A -85,B 0,C 180,E1 -9837.167,E2 -9837.167} C_VEL
LIN {X 0,Y 425.294,Z 297.507,A -85,B 0,C 180,E1 -9840.817,E2 -9840.817} C_VEL
LIN {X 0,Y 425.316,Z 297.509,A -85,B 0,C 180,E1 -9844.288,E2 -9844.288} C_VEL
LIN {X 0,Y 425.283,Z 297.506,A -85,B 0,C 180,E1 -9847.695,E2 -9847.695} C_VEL
LIN {X 0,Y 425.286,Z 297.512,A -85,B 0,C 180,E1 -9850.521,E2 -9850.521} C_VEL
LIN {X 0,Y 425.263,Z 297.508,A -85,B 0,C 180,E1 -9853.351,E2 -9853.351} C_VEL
LIN {X 0,Y 425.264,Z 297.515,A -85,B 0,C 180,E1 -9856.649,E2 -9856.649} C_VEL
LIN {X 0,Y 425.292,Z 297.504,A -85,B 0,C 180,E1 -9859.873,E2 -9859.873} C_VEL
LIN {X 0,Y 425.284,Z 297.508,A -85,B 0,C 180,E1 -9862.489,E2 -9862.489} C_VEL
LIN {X 0,Y 425.292,Z 297.504,A -85,B 0,C 180,E1 -9865.816,E2 -9865.816} C_VEL
LIN {X 0,Y 425.297,Z 297.509,A -85,B 0,C 180,E1 -9869.239,E2 -9869.239} C_VEL
LIN {X 0,Y 425.355,Z 297.496,A -85,B 0,C 180,E1 -9872.442,E2 -9872.442} C_VEL
LIN {X 0,Y 425.356,Z 297.5,A -85,B 0,C 180,E1 -9875.602,E2 -9875.602} C_VEL
LIN {X 0,Y 425.299,Z 297.503,A -85,B 0,C 180,E1 -9878.682,E2 -9878.682} C_VEL
LIN {X 0,Y 425.328,Z 297.505,A -85,B 0,C 180,E1 -9881.702,E2 -9881.702} C_VEL
LIN {X 0,Y 425.353,Z 297.496,A -85,B 0,C 180,E1 -9884.671,E2 -9884.671} C_VEL
LIN {X 0,Y 425.418,Z 297.495,A -85,B 0,C 180,E1 -9887.598,E2 -9887.598} C_VEL
LIN {X 0,Y 425.442,Z 297.488,A -85,B 0,C 180,E1 -9891.45,E2 -9891.45} C_VEL
LIN {X 0,Y 425.541,Z 297.476,A -85,B 0,C 180,E1 -9894.313,E2 -9894.313} C_VEL
LIN {X 0,Y 425.578,Z 297.476,A -85,B 0,C 180,E1 -9898.107,E2 -9898.107} C_VEL
LIN {X 0,Y 425.704,Z 297.459,A -85,B 0,C 180,E1 -9900,E2 -9900} C_VEL
LIN {X 0,Y 425.549,Z 297.473,A -85,B 0,C 180,E1 -9902.84,E2 -9902.84} C_VEL
LIN {X 0,Y 425.552,Z 297.473,A -85,B 0,C 180,E1 -9905.687,E2 -9905.687} C_VEL
LIN {X 0,Y 425.413,Z 297.495,A -85,B 0,C 180,E1 -9908.55,E2 -9908.55} C_VEL
LIN {X 0,Y 425.417,Z 297.495,A -85,B 0,C 180,E1 -9912.401,E2 -9912.401} C_VEL
LIN {X 0,Y 425.393,Z 297.495,A -85,B 0,C 180,E1 -9916.311,E2 -9916.311} C_VEL
LIN {X 0,Y 425.333,Z 297.499,A -85,B 0,C 180,E1 -9919.635,E2 -9919.635} C_VEL
LIN {X 0,Y 425.293,Z 297.506,A -85,B 0,C 180,E1 -9922.338,E2 -9922.338} C_VEL
LIN {X 0,Y 425.3,Z 297.505,A -85,B 0,C 180,E1 -9925.445,E2 -9925.445} C_VEL
LIN {X 0,Y 425.336,Z 297.501,A -85,B 0,C 180,E1 -9928.632,E2 -9928.632} C_VEL
LIN {X 0,Y 425.269,Z 297.507,A -85,B 0,C 180,E1 -9931.926,E2 -9931.926} C_VEL
LIN {X 0,Y 425.303,Z 297.51,A -85,B 0,C 180,E1 -9935.335,E2 -9935.335} C_VEL
LIN {X 0,Y 425.301,Z 297.506,A -85,B 0,C 180,E1 -9939.043,E2 -9939.043} C_VEL
LIN {X 0,Y 425.279,Z 297.506,A -85,B 0,C 180,E1 -9942.652,E2 -9942.652} C_VEL
LIN {X 0,Y 425.265,Z 297.51,A -85,B 0,C 180,E1 -9946.043,E2 -9946.043} C_VEL
LIN {X 0,Y 425.278,Z 297.506,A -85,B 0,C 180,E1 -9948.621,E2 -9948.621} C_VEL
LIN {X 0,Y 425.301,Z 297.504,A -85,B 0,C 180,E1 -9951.1,E2 -9951.1} C_VEL
LIN {X 0,Y 425.303,Z 297.503,A -85,B 0,C 180,E1 -9954.663,E2 -9954.663} C_VEL
LIN {X 0,Y 425.269,Z 297.514,A -85,B 0,C 180,E1 -9958.072,E2 -9958.072} C_VEL
LIN {X 0,Y 425.335,Z 297.499,A -85,B 0,C 180,E1 -9961.367,E2 -9961.367} C_VEL
LIN {X 0,Y 425.357,Z 297.496,A -85,B 0,C 180,E1 -9963.504,E2 -9963.504} C_VEL
LIN {X 0,Y 425.308,Z 297.505,A -85,B 0,C 180,E1 -9966.634,E2 -9966.634} C_VEL
LIN {X 0,Y 425.364,Z 297.502,A -85,B 0,C 180,E1 -9970.351,E2 -9970.351} C_VEL
LIN {X 0,Y 425.391,Z 297.492,A -85,B 0,C 180,E1 -9973.687,E2 -9973.687} C_VEL
LIN {X 0,Y 425.414,Z 297.489,A -85,B 0,C 180,E1 -9977.597,E2 -9977.597} C_VEL
LIN {X 0,Y 425.409,Z 297.494,A -85,B 0,C 180,E1 -9981.448,E2 -9981.448} C_VEL
LIN {X 0,Y 425.521,Z 297.486,A -85,B 0,C 180,E1 -9983.3,E2 -9983.3} C_VEL
LIN {X 0,Y 426.845,Z 306.237,A -85,B 0,C 180,E1 -9985.276,E2 -9985.276} C_VEL
LIN {X 0,Y 426.701,Z 312.485,A -85,B 0,C 180,E1 -9986.59,E2 -9986.59} C_VEL
LIN {X 0,Y 430.346,Z 331.738,A -85,B 0,C 180,E1 -9987.065,E2 -9987.065} C_VEL
LIN {X 0,Y 429.551,Z 399.557,A -85,B 0,C 180,E1 -9988.197,E2 -9988.197} C_VEL
LIN {X 0,Y 428.769,Z 405.405,A -85,B 0,C 180,E1 -9988.267,E2 -9988.267} C_VEL
LIN {X 0,Y 423.036,Z 423.33,A -85,B 0,C 180,E1 -9988.434,E2 -9988.434} C_VEL
LIN {X 0,Y 422.224,Z 428.097,A -85,B 0,C 180,E1 -9988.555,E2 -9988.555} C_VEL
LIN {X 0,Y 422.141,Z 430.007,A -85,B 0,C 180,E1 -9988.618,E2 -9988.618} C_VEL
LIN {X 0,Y 421.725,Z 442.278,A -85,B 0,C 180,E1 -9989.151,E2 -9989.151} C_VEL
LIN {X 0,Y 421.228,Z 454.451,A -85,B 0,C 180,E1 -9989.879,E2 -9989.879} C_VEL
LIN {X 0,Y 420.57,Z 465.337,A -85,B 0,C 180,E1 -9990.717,E2 -9990.717} C_VEL
LIN {X 0,Y 419.829,Z 476.441,A -85,B 0,C 180,E1 -9991.797,E2 -9991.797} C_VEL
LIN {X 0,Y 419.262,Z 485.409,A -85,B 0,C 180,E1 -9992.881,E2 -9992.881} C_VEL
LIN {X 0,Y 418.544,Z 495.151,A -85,B 0,C 180,E1 -9994.332,E2 -9994.332} C_VEL
LIN {X 0,Y 418.018,Z 502.94,A -85,B 0,C 180,E1 -9995.788,E2 -9995.788} C_VEL
LIN {X 0,Y 417.748,Z 509.253,A -85,B 0,C 180,E1 -9997.273,E2 -9997.273} C_VEL
LIN {X 0,Y 417.424,Z 514.124,A -85,B 0,C 180,E1 -9998.714,E2 -9998.714} C_VEL
LIN {X 0,Y 417.254,Z 517.953,A -85,B 0,C 180,E1 -10000.185,E2 -10000.185} C_VEL
LIN {X 0,Y 417.035,Z 521.535,A -85,B 0,C 180,E1 -10002.196,E2 -10002.196} C_VEL
LIN {X 0,Y 416.95,Z 522.985,A -85,B 0,C 180,E1 -10003.648,E2 -10003.648} C_VEL
LIN {X 0,Y 416.917,Z 523.448,A -85,B 0,C 180,E1 -10004.645,E2 -10004.645} C_VEL
LIN {X 0,Y 416.954,Z 523.4,A -85,B 0,C 180,E1 -10006.103,E2 -10006.103} C_VEL
LIN {X 0,Y 416.997,Z 522.35,A -85,B 0,C 180,E1 -10007.658,E2 -10007.658} C_VEL
LIN {X 0,Y 417.198,Z 519.96,A -85,B 0,C 180,E1 -10009.377,E2 -10009.377} C_VEL
LIN {X 0,Y 417.464,Z 515.936,A -85,B 0,C 180,E1 -10011.218,E2 -10011.218} C_VEL
LIN {X 0,Y 417.798,Z 511.269,A -85,B 0,C 180,E1 -10012.76,E2 -10012.76} C_VEL
LIN {X 0,Y 418.3,Z 505.201,A -85,B 0,C 180,E1 -10014.306,E2 -10014.306} C_VEL
LIN {X 0,Y 418.92,Z 497.474,A -85,B 0,C 180,E1 -10015.859,E2 -10015.859} C_VEL
LIN {X 0,Y 419.617,Z 489.348,A -85,B 0,C 180,E1 -10017.176,E2 -10017.176} C_VEL
LIN {X 0,Y 420.436,Z 479.64,A -85,B 0,C 180,E1 -10018.449,E2 -10018.449} C_VEL
LIN {X 0,Y 421.196,Z 468.922,A -85,B 0,C 180,E1 -10019.577,E2 -10019.577} C_VEL
LIN {X 0,Y 422.013,Z 457.579,A -85,B 0,C 180,E1 -10020.524,E2 -10020.524} C_VEL
LIN {X 0,Y 422.676,Z 445.453,A -85,B 0,C 180,E1 -10021.304,E2 -10021.304} C_VEL
LIN {X 0,Y 423.277,Z 432.292,A -85,B 0,C 180,E1 -10021.917,E2 -10021.917} C_VEL
LIN {X 0,Y 423.622,Z 419.77,A -85,B 0,C 180,E1 -10022.309,E2 -10022.309} C_VEL
LIN {X 0,Y 424.699,Z 331.872,A -85,B 0,C 180,E1 -10023.849,E2 -10023.849} C_VEL
LIN {X 0,Y 420.765,Z 314.432,A -85,B 0,C 180,E1 -10024.381,E2 -10024.381} C_VEL
LIN {X 0,Y 420.341,Z 312.63,A -85,B 0,C 180,E1 -10024.441,E2 -10024.441} C_VEL
LIN {X 0,Y 420.298,Z 308.45,A -85,B 0,C 180,E1 -10025.35,E2 -10025.35} C_VEL
LIN {X 0,Y 418.224,Z 298.392,A -85,B 0,C 180,E1 -10027.747,E2 -10027.747} C_VEL
LIN {X 0,Y 418.196,Z 298.391,A -85,B 0,C 180,E1 -10030.949,E2 -10030.949} C_VEL
LIN {X 0,Y 418.19,Z 298.394,A -85,B 0,C 180,E1 -10033.727,E2 -10033.727} C_VEL
LIN {X 0,Y 418.19,Z 298.386,A -85,B 0,C 180,E1 -10036.446,E2 -10036.446} C_VEL
LIN {X 0,Y 418.195,Z 298.393,A -85,B 0,C 180,E1 -10039.132,E2 -10039.132} C_VEL
LIN {X 0,Y 418.221,Z 298.389,A -85,B 0,C 180,E1 -10042.774,E2 -10042.774} C_VEL
LIN {X 0,Y 418.234,Z 298.387,A -85,B 0,C 180,E1 -10046.322,E2 -10046.322} C_VEL
LIN {X 0,Y 418.229,Z 298.39,A -85,B 0,C 180,E1 -10049.727,E2 -10049.727} C_VEL
LIN {X 0,Y 418.23,Z 298.385,A -85,B 0,C 180,E1 -10053.018,E2 -10053.018} C_VEL
LIN {X 0,Y 418.259,Z 298.386,A -85,B 0,C 180,E1 -10056.217,E2 -10056.217} C_VEL
LIN {X 0,Y 418.235,Z 298.38,A -85,B 0,C 180,E1 -10059.336,E2 -10059.336} C_VEL
LIN {X 0,Y 418.271,Z 298.378,A -85,B 0,C 180,E1 -10062.396,E2 -10062.396} C_VEL
LIN {X 0,Y 418.286,Z 298.378,A -85,B 0,C 180,E1 -10065.403,E2 -10065.403} C_VEL
LIN {X 0,Y 418.301,Z 298.375,A -85,B 0,C 180,E1 -10068.369,E2 -10068.369} C_VEL
LIN {X 0,Y 418.382,Z 298.365,A -85,B 0,C 180,E1 -10071.305,E2 -10071.305} C_VEL
LIN {X 0,Y 418.482,Z 298.352,A -85,B 0,C 180,E1 -10074.217,E2 -10074.217} C_VEL
LIN {X 0,Y 418.528,Z 298.345,A -85,B 0,C 180,E1 -10078.076,E2 -10078.076} C_VEL
LIN {X 0,Y 418.657,Z 298.331,A -85,B 0,C 180,E1 -10080,E2 -10080} C_VEL
LIN {X 0,Y 418.487,Z 298.347,A -85,B 0,C 180,E1 -10082.888,E2 -10082.888} C_VEL
LIN {X 0,Y 418.477,Z 298.356,A -85,B 0,C 180,E1 -10086.752,E2 -10086.752} C_VEL
LIN {X 0,Y 418.386,Z 298.362,A -85,B 0,C 180,E1 -10088.696,E2 -10088.696} C_VEL
LIN {X 0,Y 418.303,Z 298.375,A -85,B 0,C 180,E1 -10091.632,E2 -10091.632} C_VEL
LIN {X 0,Y 418.289,Z 298.373,A -85,B 0,C 180,E1 -10094.598,E2 -10094.598} C_VEL
LIN {X 0,Y 418.275,Z 298.377,A -85,B 0,C 180,E1 -10097.605,E2 -10097.605} C_VEL
LIN {X 0,Y 418.237,Z 298.386,A -85,B 0,C 180,E1 -10100.664,E2 -10100.664} C_VEL
LIN {X 0,Y 418.276,Z 298.375,A -85,B 0,C 180,E1 -10103.782,E2 -10103.782} C_VEL
LIN {X 0,Y 418.298,Z 298.379,A -85,B 0,C 180,E1 -10107.072,E2 -10107.072} C_VEL
LIN {X 0,Y 418.253,Z 298.383,A -85,B 0,C 180,E1 -10110.272,E2 -10110.272} C_VEL
LIN {X 0,Y 418.239,Z 298.389,A -85,B 0,C 180,E1 -10113.678,E2 -10113.678} C_VEL
LIN {X 0,Y 418.238,Z 298.389,A -85,B 0,C 180,E1 -10117.225,E2 -10117.225} C_VEL
LIN {X 0,Y 418.256,Z 298.387,A -85,B 0,C 180,E1 -10119.682,E2 -10119.682} C_VEL
LIN {X 0,Y 418.239,Z 298.383,A -85,B 0,C 180,E1 -10122.325,E2 -10122.325} C_VEL
